    TEXT311 : BOOL ;	//TEXT N.311
    TEXT312 : BOOL ;	//TEXT N.312
    TEXT329 : BOOL ;	//TEXT N.329
    TEXT330 : BOOL ;	//TEXT N.330
    TEXT331 : BOOL ;	//TEXT N.331
    TEXT332 : BOOL ;	//TEXT N.332
    TEXT333 : BOOL ;	//TEXT N.333
    TEXT334 : BOOL ;	//TEXT N.334
    TEXT335 : BOOL ;	//TEXT N.335
    TEXT336 : BOOL ;	//TEXT N.336
    TEXT321 : BOOL ;	//TEXT N.321
    TEXT322 : BOOL ;	//TEXT N.322
    TEXT323 : BOOL ;	//TEXT N.323
    TEXT324 : BOOL ;	//TEXT N.324
    TEXT325 : BOOL ;	//TEXT N.325
    TEXT326 : BOOL ;	//TEXT N.326
    TEXT327 : BOOL ;	//TEXT N.327
    TEXT328 : BOOL ;	//TEXT N.328
    TEXT345 : BOOL ;	//TEXT N.345
    TEXT346 : BOOL ;	//TEXT N.346
    TEXT347 : BOOL ;	//TEXT N.347
    TEXT348 : BOOL ;	//TEXT N.348
    TEXT349 : BOOL ;	//TEXT N.349
    TEXT350 : BOOL ;	//TEXT N.350
    TEXT351 : BOOL ;	//TEXT N.351
    TEXT352 : BOOL ;	//TEXT N.352
    TEXT337 : BOOL ;	//TEXT N.337
    TEXT338 : BOOL ;	//TEXT N.338
    TEXT339 : BOOL ;	//TEXT N.339
    TEXT340 : BOOL ;	//TEXT N.340
    TEXT341 : BOOL ;	//TEXT N.341
    TEXT342 : BOOL ;	//TEXT N.342
    TEXT343 : BOOL ;	//TEXT N.343
    TEXT344 : BOOL ;	//TEXT N.344
    TEXT361 : BOOL ;	//TEXT N.361
    TEXT362 : BOOL ;	//TEXT N.362
    TEXT363 : BOOL ;	//TEXT N.363
    TEXT364 : BOOL ;	//TEXT N.364
    TEXT365 : BOOL ;	//TEXT N.365
    TEXT366 : BOOL ;	//TEXT N.366
    TEXT367 : BOOL ;	//TEXT N.367
    TEXT368 : BOOL ;	//TEXT N.368
    TEXT353 : BOOL ;	//TEXT N.353
    TEXT354 : BOOL ;	//TEXT N.354
    TEXT355 : BOOL ;	//TEXT N.355
    TEXT356 : BOOL ;	//TEXT N.356
    TEXT357 : BOOL ;	//TEXT N.357
    TEXT358 : BOOL ;	//TEXT N.358
    TEXT359 : BOOL ;	//TEXT N.359
    TEXT360 : BOOL ;	//TEXT N.360
    TEXT377 : BOOL ;	//TEXT N.377
    TEXT378 : BOOL ;	//TEXT N.378
    TEXT379 : BOOL ;	//TEXT N.379
    TEXT380 : BOOL ;	//TEXT N.380
    TEXT381 : BOOL ;	//TEXT N.381
    TEXT382 : BOOL ;	//TEXT N.382
    TEXT383 : BOOL ;	//TEXT N.383
    TEXT384 : BOOL ;	//TEXT N.384
    TEXT369 : BOOL ;	//TEXT N.369
    TEXT370 : BOOL ;	//TEXT N.370
    TEXT371 : BOOL ;	//TEXT N.371
    TEXT372 : BOOL ;	//TEXT N.372
    TEXT373 : BOOL ;	//TEXT N.373
    TEXT374 : BOOL ;	//TEXT N.374
    TEXT375 : BOOL ;	//TEXT N.375
    TEXT376 : BOOL ;	//TEXT N.376
    TEXT393 : BOOL ;	//TEXT N.393
    TEXT394 : BOOL ;	//TEXT N.394
    TEXT395 : BOOL ;	//TEXT N.395
    TEXT396 : BOOL ;	//TEXT N.396
    TEXT397 : BOOL ;	//TEXT N.397
    TEXT398 : BOOL ;	//TEXT N.398
    TEXT399 : BOOL ;	//TEXT N.399
    TEXT400 : BOOL ;	//TEXT N.400
    TEXT385 : BOOL ;	//TEXT N.385
    TEXT386 : BOOL ;	//TEXT N.386
    TEXT387 : BOOL ;	//TEXT N.387
    TEXT388 : BOOL ;	//TEXT N.388
    TEXT389 : BOOL ;	//TEXT N.389
    TEXT390 : BOOL ;	//TEXT N.390
    TEXT391 : BOOL ;	//TEXT N.391
    TEXT392 : BOOL ;	//TEXT N.392
    TEXT409 : BOOL ;	//TEXT N.409
    TEXT410 : BOOL ;	//TEXT N.410
    TEXT411 : BOOL ;	//TEXT N.411
    TEXT412 : BOOL ;	//TEXT N.412
    TEXT413 : BOOL ;	//TEXT N.413
    TEXT414 : BOOL ;	//TEXT N.414
    TEXT415 : BOOL ;	//TEXT N.415
    TEXT416 : BOOL ;	//TEXT N.416
    TEXT401 : BOOL ;	//TEXT N.401
    TEXT402 : BOOL ;	//TEXT N.402
    TEXT403 : BOOL ;	//TEXT N.403
    TEXT404 : BOOL ;	//TEXT N.404
    TEXT405 : BOOL ;	//TEXT N.405
    TEXT406 : BOOL ;	//TEXT N.406
    TEXT407 : BOOL ;	//TEXT N.407
    TEXT408 : BOOL ;	//TEXT N.408
    TEXT425 : BOOL ;	//TEXT N.425
    TEXT426 : BOOL ;	//TEXT N.426
    TEXT427 : BOOL ;	//TEXT N.427
    TEXT428 : BOOL ;	//TEXT N.428
    TEXT429 : BOOL ;	//TEXT N.429
    TEXT430 : BOOL ;	//TEXT N.430
    TEXT431 : BOOL ;	//TEXT N.431
    TEXT432 : BOOL ;	//TEXT N.432
    TEXT417 : BOOL ;	//TEXT N.417
    TEXT418 : BOOL ;	//TEXT N.418
    TEXT419 : BOOL ;	//TEXT N.419
    TEXT420 : BOOL ;	//TEXT N.420
    TEXT421 : BOOL ;	//TEXT N.421
    TEXT422 : BOOL ;	//TEXT N.422
    TEXT423 : BOOL ;	//TEXT N.423
    TEXT424 : BOOL ;	//TEXT N.424
    TEXT441 : BOOL ;	//TEXT N.441
    TEXT442 : BOOL ;	//TEXT N.442
    TEXT443 : BOOL ;	//TEXT N.443
    TEXT444 : BOOL ;	//TEXT N.444
    TEXT445 : BOOL ;	//TEXT N.445
    TEXT446 : BOOL ;	//TEXT N.446
    TEXT447 : BOOL ;	//TEXT N.447
    TEXT448 : BOOL ;	//TEXT N.448
    TEXT433 : BOOL ;	//TEXT N.433
    TEXT434 : BOOL ;	//TEXT N.434
    TEXT435 : BOOL ;	//TEXT N.435
    TEXT436 : BOOL ;	//TEXT N.436
    TEXT437 : BOOL ;	//TEXT N.437
    TEXT438 : BOOL ;	//TEXT N.438
    TEXT439 : BOOL ;	//TEXT N.439
    TEXT440 : BOOL ;	//TEXT N.440
    TEXT457 : BOOL ;	//TEXT N.457
    TEXT458 : BOOL ;	//TEXT N.458
    TEXT459 : BOOL ;	//TEXT N.459
    TEXT460 : BOOL ;	//TEXT N.460
    TEXT461 : BOOL ;	//TEXT N.461
    TEXT462 : BOOL ;	//TEXT N.462
    TEXT463 : BOOL ;	//TEXT N.463
    TEXT464 : BOOL ;	//TEXT N.464
    TEXT449 : BOOL ;	//TEXT N.449
    TEXT450 : BOOL ;	//TEXT N.450
    TEXT451 : BOOL ;	//TEXT N.451
    TEXT452 : BOOL ;	//TEXT N.452
    TEXT453 : BOOL ;	//TEXT N.453
    TEXT454 : BOOL ;	//TEXT N.454
    TEXT455 : BOOL ;	//TEXT N.455
    TEXT456 : BOOL ;	//TEXT N.456
    TEXT473 : BOOL ;	//TEXT N.473
    TEXT474 : BOOL ;	//TEXT N.474
    TEXT475 : BOOL ;	//TEXT N.475
    TEXT476 : BOOL ;	//TEXT N.476
    TEXT477 : BOOL ;	//TEXT N.477
    TEXT478 : BOOL ;	//TEXT N.478
    TEXT479 : BOOL ;	//TEXT N.479
    TEXT480 : BOOL ;	//TEXT N.480
    TEXT465 : BOOL ;	//TEXT N.465
    TEXT466 : BOOL ;	//TEXT N.466
    TEXT467 : BOOL ;	//TEXT N.467
    TEXT468 : BOOL ;	//TEXT N.468
    TEXT469 : BOOL ;	//TEXT N.469
    TEXT470 : BOOL ;	//TEXT N.470
    TEXT471 : BOOL ;	//TEXT N.471
    TEXT472 : BOOL ;	//TEXT N.472
    TEXT489 : BOOL ;	//TEXT N.489
    TEXT490 : BOOL ;	//TEXT N.490
    TEXT491 : BOOL ;	//TEXT N.491
    TEXT492 : BOOL ;	//TEXT N.492
    TEXT493 : BOOL ;	//TEXT N.493
    TEXT494 : BOOL ;	//TEXT N.494
    TEXT495 : BOOL ;	//TEXT N.495
    TEXT496 : BOOL ;	//TEXT N.496
    TEXT481 : BOOL ;	//TEXT N.481
    TEXT482 : BOOL ;	//TEXT N.482
    TEXT483 : BOOL ;	//TEXT N.483
    TEXT484 : BOOL ;	//TEXT N.484
    TEXT485 : BOOL ;	//TEXT N.485
    TEXT486 : BOOL ;	//TEXT N.486
    TEXT487 : BOOL ;	//TEXT N.487
    TEXT488 : BOOL ;	//TEXT N.488
    TEXT505 : BOOL ;	//TEXT N.505
    TEXT506 : BOOL ;	//TEXT N.506
    TEXT507 : BOOL ;	//TEXT N.507
    TEXT508 : BOOL ;	//TEXT N.508
    TEXT509 : BOOL ;	//TEXT N.509
    TEXT510 : BOOL ;	//TEXT N.510
    TEXT511 : BOOL ;	//TEXT N.511
    TEXT512 : BOOL ;	//TEXT N.512
    TEXT497 : BOOL ;	//TEXT N.497
    TEXT498 : BOOL ;	//TEXT N.498
    TEXT499 : BOOL ;	//TEXT N.499
    TEXT500 : BOOL ;	//TEXT N.500
    TEXT501 : BOOL ;	//TEXT N.501
    TEXT502 : BOOL ;	//TEXT N.502
    TEXT503 : BOOL ;	//TEXT N.503
    TEXT504 : BOOL ;	//TEXT N.504
    TEXT521 : BOOL ;	//TEXT N.521
    TEXT522 : BOOL ;	//TEXT N.522
    TEXT523 : BOOL ;	//TEXT N.523
    TEXT524 : BOOL ;	//TEXT N.524
    TEXT525 : BOOL ;	//TEXT N.525
    TEXT526 : BOOL ;	//TEXT N.526
    TEXT527 : BOOL ;	//TEXT N.527
    TEXT528 : BOOL ;	//TEXT N.528
    TEXT513 : BOOL ;	//TEXT N.513
    TEXT514 : BOOL ;	//TEXT N.514
    TEXT515 : BOOL ;	//TEXT N.515
    TEXT516 : BOOL ;	//TEXT N.516
    TEXT517 : BOOL ;	//TEXT N.517
    TEXT518 : BOOL ;	//TEXT N.518
    TEXT519 : BOOL ;	//TEXT N.519
    TEXT520 : BOOL ;	//TEXT N.520
    TEXT537 : BOOL ;	//TEXT N.537
    TEXT538 : BOOL ;	//TEXT N.538
    TEXT539 : BOOL ;	//TEXT N.539
    TEXT540 : BOOL ;	//TEXT N.540
    TEXT541 : BOOL ;	//TEXT N.541
    TEXT542 : BOOL ;	//TEXT N.542
    TEXT543 : BOOL ;	//TEXT N.543
    TEXT544 : BOOL ;	//TEXT N.544
    TEXT529 : BOOL ;	//TEXT N.529
    TEXT530 : BOOL ;	//TEXT N.530
    TEXT531 : BOOL ;	//TEXT N.531
    TEXT532 : BOOL ;	//TEXT N.532
    TEXT533 : BOOL ;	//TEXT N.533
    TEXT534 : BOOL ;	//TEXT N.534
    TEXT535 : BOOL ;	//TEXT N.535
    TEXT536 : BOOL ;	//TEXT N.536
    TEXT553 : BOOL ;	//TEXT N.553
    TEXT554 : BOOL ;	//TEXT N.554
    TEXT555 : BOOL ;	//TEXT N.555
    TEXT556 : BOOL ;	//TEXT N.556
    TEXT557 : BOOL ;	//TEXT N.557
    TEXT558 : BOOL ;	//TEXT N.558
    TEXT559 : BOOL ;	//TEXT N.559
    TEXT560 : BOOL ;	//TEXT N.560
    TEXT545 : BOOL ;	//TEXT N.545
    TEXT546 : BOOL ;	//TEXT N.546
    TEXT547 : BOOL ;	//TEXT N.547
    TEXT548 : BOOL ;	//TEXT N.548
    TEXT549 : BOOL ;	//TEXT N.549
    TEXT550 : BOOL ;	//TEXT N.550
    TEXT551 : BOOL ;	//TEXT N.551
    TEXT552 : BOOL ;	//TEXT N.552
    TEXT569 : BOOL ;	//TEXT N.569
    TEXT570 : BOOL ;	//TEXT N.570
    TEXT571 : BOOL ;	//TEXT N.571
    TEXT572 : BOOL ;	//TEXT N.572
    TEXT573 : BOOL ;	//TEXT N.573
    TEXT574 : BOOL ;	//TEXT N.574
    TEXT575 : BOOL ;	//TEXT N.575
    TEXT576 : BOOL ;	//TEXT N.576
    TEXT561 : BOOL ;	//TEXT N.561
    TEXT562 : BOOL ;	//TEXT N.562
    TEXT563 : BOOL ;	//TEXT N.563
    TEXT564 : BOOL ;	//TEXT N.564
    TEXT565 : BOOL ;	//TEXT N.565
    TEXT566 : BOOL ;	//TEXT N.566
    TEXT567 : BOOL ;	//TEXT N.567
    TEXT568 : BOOL ;	//TEXT N.568
    TEXT585 : BOOL ;	//TEXT N.585
    TEXT586 : BOOL ;	//TEXT N.586
    TEXT587 : BOOL ;	//TEXT N.587
    TEXT588 : BOOL ;	//TEXT N.588
    TEXT589 : BOOL ;	//TEXT N.589
    TEXT590 : BOOL ;	//TEXT N.590
    TEXT591 : BOOL ;	//TEXT N.591
    TEXT592 : BOOL ;	//TEXT N.592
    TEXT577 : BOOL ;	//TEXT N.577
    TEXT578 : BOOL ;	//TEXT N.578
    TEXT579 : BOOL ;	//TEXT N.579
    TEXT580 : BOOL ;	//TEXT N.580
    TEXT581 : BOOL ;	//TEXT N.581
    TEXT582 : BOOL ;	//TEXT N.582
    TEXT583 : BOOL ;	//TEXT N.583
    TEXT584 : BOOL ;	//TEXT N.584
    TEXT601 : BOOL ;	//TEXT N.601
    TEXT602 : BOOL ;	//TEXT N.602
    TEXT603 : BOOL ;	//TEXT N.603
    TEXT604 : BOOL ;	//TEXT N.604
    TEXT605 : BOOL ;	//TEXT N.605
    TEXT606 : BOOL ;	//TEXT N.606
    TEXT607 : BOOL ;	//TEXT N.607
    TEXT608 : BOOL ;	//TEXT N.608
    TEXT593 : BOOL ;	//TEXT N.593
    TEXT594 : BOOL ;	//TEXT N.594
    TEXT595 : BOOL ;	//TEXT N.595
    TEXT596 : BOOL ;	//TEXT N.596
    TEXT597 : BOOL ;	//TEXT N.597
    TEXT598 : BOOL ;	//TEXT N.598
    TEXT599 : BOOL ;	//TEXT N.599
    TEXT600 : BOOL ;	//TEXT N.600
    TEXT617 : BOOL ;	//TEXT N.617
    TEXT618 : BOOL ;	//TEXT N.618
    TEXT619 : BOOL ;	//TEXT N.619
    TEXT620 : BOOL ;	//TEXT N.620
    TEXT621 : BOOL ;	//TEXT N.621
    TEXT622 : BOOL ;	//TEXT N.622
    TEXT623 : BOOL ;	//TEXT N.623
    TEXT624 : BOOL ;	//TEXT N.624
    TEXT609 : BOOL ;	//TEXT N.609
    TEXT610 : BOOL ;	//TEXT N.610
    TEXT611 : BOOL ;	//TEXT N.611
    TEXT612 : BOOL ;	//TEXT N.612
    TEXT613 : BOOL ;	//TEXT N.613
    TEXT614 : BOOL ;	//TEXT N.614
    TEXT615 : BOOL ;	//TEXT N.615
    TEXT616 : BOOL ;	//TEXT N.616
    TEXT633 : BOOL ;	//TEXT N.633
    TEXT634 : BOOL ;	//TEXT N.634
    TEXT635 : BOOL ;	//TEXT N.635
    TEXT636 : BOOL ;	//TEXT N.636
    TEXT637 : BOOL ;	//TEXT N.637
    TEXT638 : BOOL ;	//TEXT N.638
    TEXT639 : BOOL ;	//TEXT N.639
    TEXT640 : BOOL ;	//TEXT N.640
    TEXT625 : BOOL ;	//TEXT N.625
    TEXT626 : BOOL ;	//TEXT N.626
    TEXT627 : BOOL ;	//TEXT N.627
    TEXT628 : BOOL ;	//TEXT N.628
    TEXT629 : BOOL ;	//TEXT N.629
    TEXT630 : BOOL ;	//TEXT N.630
    TEXT631 : BOOL ;	//TEXT N.631
    TEXT632 : BOOL ;	//TEXT N.632
   END_STRUCT ;
   PaginaDaVisualizzare : INT ;	//Number of page to display
   PaginaPrecedenteSetup : INT ;	//Number of page displayed before "Setup" page
   NumeroComandoManuale : INT ;	//Number of manual command
   BoschProgramManuale : BYTE ;	//Number of program of screwdriver in manual mode
   ServiceAsseSelezionato : BYTE ;	//Axis selected for movement in service mode (0=X; 1=Y; 2=Z; 3=C; 4=P)
   ServiceTipoJog : BYTE ;	//Kind of jog movement in service mode (0=continue; 1=incremental)
   ServiceFieldsDisplayed : BYTE ;	//Identify the fields to be displayed in service page
   TypePointTeachIn : BYTE ;	//Kind of screw in teach-in mode
   PointWeldingTeachIn : BYTE ;	//Identification of the screw in tech-in mode
   TeachInFieldsDisplayed : STRUCT 	//Identify the fields to be displayed in teach-in page
    Punto1Saldatura : BOOL ;
    Punto2Saldatura : BOOL ;
    Punto3Saldatura : BOOL ;
    Punto4Saldatura : BOOL ;
    Punto5Saldatura : BOOL ;
    Punto6Saldatura : BOOL ;
    Punto7Saldatura : BOOL ;
    Punto8Saldatura : BOOL ;
    Punto9Saldatura : BOOL ;
    Punto10Saldatura : BOOL ;
    Punto11Saldatura : BOOL ;
    Punto12Saldatura : BOOL ;
    Punto13Saldatura : BOOL ;
    PuntoVisione : BOOL ;
    Riserva1 : BOOL ;
    Riserva2 : BOOL ;
   END_STRUCT ;
   Target_Inc : DINT ;	//Target for the incremental movement
  END_STRUCT ;	
BEGIN
END_DATA_BLOCK

DATA_BLOCK "Timer"	// DB 20
VERSION : 0.1
  STRUCT
   TmrOutGas : S5TIME  := S5T#1M;
   TmrIgnition : S5TIME  := S5T#20S;
   TmrDelayWelding : S5TIME  := S5T#300MS;
   time1 : S5TIME ;
   time11 : S5TIME ;
   time12 : S5TIME ;
   time13 : S5TIME ;
   time14 : S5TIME ;
   time15 : S5TIME ;
   time16 : S5TIME ;
   time17 : S5TIME ;
   time18 : S5TIME ;
   time19 : S5TIME ;
   time110 : S5TIME ;
   time111 : S5TIME ;
   time112 : S5TIME ;
   time113 : S5TIME ;
   time114 : S5TIME ;
   time115 : S5TIME ;
   time116 : S5TIME ;
   Override : INT  := 20;
   riserva : INT ;
   riserva2 : INT ;
   Comp01_OK : BOOL ;
   Comp02_OK : BOOL ;
   Comp03_OK : BOOL ;
   Comp04_OK : BOOL ;
   Comp05_OK : BOOL ;
   Comp06_OK : BOOL ;
   Comp07_OK : BOOL ;
   Comp08_OK : BOOL ;
   Comp09_OK : BOOL ;
   Comp10_OK : BOOL ;
   Comp11_OK : BOOL ;
   Comp12_OK : BOOL ;
   Comp13_OK : BOOL ;
   Comp14_OK : BOOL ;
   Comp15_OK : BOOL ;
   Comp16_OK : BOOL ;
   OffsetX : DINT ;
   OffsetY : DINT ;
   okAletta1 : BOOL ;
   okAletta2 : BOOL ;
   okAletta3 : BOOL ;
   okAletta4 : BOOL ;
   okAletta5 : BOOL ;
   okAletta6 : BOOL ;
   okAletta7 : BOOL ;
   okAletta8 : BOOL ;
   okAletta9 : BOOL ;
   okAletta10 : BOOL ;
   okAletta11 : BOOL ;
   okAletta12 : BOOL ;
   okAletta13 : BOOL ;
   okAletta14 : BOOL ;
   okAletta15 : BOOL ;
   okAletta16 : BOOL ;
   okAletta17 : BOOL ;
   okAletta18 : BOOL ;
   okAletta19 : BOOL ;
   okAletta20 : BOOL ;
   CheckComponent : BOOL  := TRUE;	//Check component with tool 1 --> Disable ; 0 --> Enable
   CheckTelec : BOOL ;	//Check Component with Omron 1 --> Disable ; 0 --> Enable
   Check1 : BOOL ;
   Check2 : BOOL ;
   okAletta1_PP : BOOL ;
   okAletta2_PP : BOOL ;
   okAletta3_PP : BOOL ;
   okAletta4_PP : BOOL ;
   okAletta5_PP : BOOL ;
   okAletta6_PP : BOOL ;
   okAletta7_PP : BOOL ;
   okAletta8_PP : BOOL ;
   okAletta9_PP : BOOL ;
   okAletta10_PP : BOOL ;
   okAletta11_PP : BOOL ;
   okAletta12_PP : BOOL ;
   okAletta13_PP : BOOL ;
   okAletta14_PP : BOOL ;
   okAletta15_PP : BOOL ;
   okAletta16_PP : BOOL ;
   okAletta17_PP : BOOL ;
   okAletta18_PP : BOOL ;
   okAletta19_PP : BOOL ;
   okAletta20_PP : BOOL ;
   NumberVane : INT ;
  END_STRUCT ;	
BEGIN
   TmrOutGas := S5T#1M;
   TmrIgnition := S5T#20S;
   TmrDelayWelding := S5T#300MS;
   Override := 100;
   OffsetX := L#350;
   OffsetY := L#400;
END_DATA_BLOCK

DATA_BLOCK "DBWork"	// DB 21
TITLE = Recipe of part in production
AUTHOR : Coletti
VERSION : 0.1
  STRUCT
   Famiglia : BYTE  := B#16#2;	//Type of family of product(2=Step2; 3=Step3)
   Turbo : BYTE  := B#16#1;	//Type of product
   Portapezzo1 : INT  := 1;	//Code of work rest 1
   Portapezzo2 : INT  := 1;	//Code of work rest 2
   TempoSaldatura : ARRAY  [1 .. 20 ] OF STRUCT
    Tempo : S5TIME  := S5T#1S;
   END_STRUCT ;
   CoordSaldatura : ARRAY  [1 .. 20 ] OF //Coordinates of points
   STRUCT
    X1 : DINT ;	//X coordinate of point
    Y1 : DINT ;	//Y coordinate of point
    X2 : DINT ;
    Y2 : DINT ;
   END_STRUCT ;
   EnableTelecamera : BOOL  := TRUE;
   PP : ARRAY  [1 .. 2 ] OF STRUCT
    Vuoto : BOOL ;
    Caricato : BOOL ;
    Bloccato : BOOL ;
    Fuori : BOOL ;
    Dentro : BOOL ;
    InLavorazione : BOOL ;
    Lavorato : BOOL ;
    Buono : BOOL ;
    Scarto : BOOL ;
    NumSaldaturaAtt : INT ;
   END_STRUCT ;
   NumeroAnomalie : DINT ;
   NumeroPezziProd : DINT ;
   NumeroSaldature : INT ;
   Riserva : DINT ;	//position X for camera check
   Riserva1 : DINT ;	//position Y for camera check
   RotationTable : BOOL ;	//angle rotation 1-->PP1 on welding; 0-->PP2 on Welding
   PointCamCheck : ARRAY  [1 .. 10 ] OF STRUCT
    x : DINT ;
    y : DINT ;
   END_STRUCT ;
  END_STRUCT ;	
BEGIN
   Famiglia := B#16#2;
   Turbo := B#16#1;
   Portapezzo1 := 1;
   Portapezzo2 := 1;
   TempoSaldatura[1].Tempo := S5T#1S;
   TempoSaldatura[2].Tempo := S5T#2S;
   TempoSaldatura[3].Tempo := S5T#1S;
   TempoSaldatura[4].Tempo := S5T#1S;
   TempoSaldatura[5].Tempo := S5T#1S;
   TempoSaldatura[6].Tempo := S5T#1S;
   TempoSaldatura[7].Tempo := S5T#1S;
   TempoSaldatura[8].Tempo := S5T#1S;
   TempoSaldatura[9].Tempo := S5T#1S;
   TempoSaldatura[10].Tempo := S5T#1S;
   TempoSaldatura[11].Tempo := S5T#1S;
   TempoSaldatura[12].Tempo := S5T#1S;
   TempoSaldatura[13].Tempo := S5T#1S;
   TempoSaldatura[14].Tempo := S5T#1S;
   TempoSaldatura[15].Tempo := S5T#1S;
   TempoSaldatura[16].Tempo := S5T#1S;
   TempoSaldatura[17].Tempo := S5T#1S;
   TempoSaldatura[18].Tempo := S5T#1S;
   TempoSaldatura[19].Tempo := S5T#1S;
   TempoSaldatura[20].Tempo := S5T#1S;
   CoordSaldatura[1].X1 := L#-60766;
   CoordSaldatura[1].Y1 := L#-86096;
   CoordSaldatura[1].X2 := L#-60406;
   CoordSaldatura[1].Y2 := L#-86246;
   CoordSaldatura[2].X1 := L#-46600;
   CoordSaldatura[2].Y1 := L#-81431;
   CoordSaldatura[2].X2 := L#-46422;
   CoordSaldatura[2].Y2 := L#-81523;
   CoordSaldatura[3].X1 := L#-29709;
   CoordSaldatura[3].Y1 := L#-81739;
   CoordSaldatura[3].X2 := L#-29405;
   CoordSaldatura[3].Y2 := L#-81809;
   CoordSaldatura[4].X1 := L#-16402;
   CoordSaldatura[4].Y1 := L#-86931;
   CoordSaldatura[4].X2 := L#-116220;
   CoordSaldatura[4].Y2 := L#-86961;
   CoordSaldatura[5].X1 := L#-11762;
   CoordSaldatura[5].Y1 := L#-95066;
   CoordSaldatura[5].X2 := L#-11500;
   CoordSaldatura[5].Y2 := L#-95199;
   CoordSaldatura[6].X1 := L#-17500;
   CoordSaldatura[6].Y1 := L#-102971;
   CoordSaldatura[6].X2 := L#-17415;
   CoordSaldatura[6].Y2 := L#-103088;
   CoordSaldatura[7].X1 := L#-31505;
   CoordSaldatura[7].Y1 := L#-107714;
   CoordSaldatura[7].X2 := L#-31400;
   CoordSaldatura[7].Y2 := L#-108200;
   CoordSaldatura[8].X1 := L#-48449;
   CoordSaldatura[8].Y1 := L#-107375;
   CoordSaldatura[8].X2 := L#-48367;
   CoordSaldatura[8].Y2 := L#-107501;
   CoordSaldatura[9].X1 := L#-61760;
   CoordSaldatura[9].Y1 := L#-102188;
   CoordSaldatura[9].X2 := L#-61561;
   CoordSaldatura[9].Y2 := L#-102300;
   CoordSaldatura[10].X1 := L#-66400;
   CoordSaldatura[10].Y1 := L#-94028;
   CoordSaldatura[10].Y2 := L#-94249;
   EnableTelecamera := TRUE;
END_DATA_BLOCK

DATA_BLOCK "coordinate"	// DB 22
VERSION : 0.1
  STRUCT
   CoordSaldaturaPP1 : ARRAY  [1 .. 20 ] OF //Coordinates of points
   STRUCT
    X1 : DINT ;	//X coordinate of point PP1
    Y1 : DINT ;	//Y coordinate of point PP1
    X2 : DINT ;
    Y2 : DINT ;
   END_STRUCT ;
   CoordSaldaturaPP2 : ARRAY  [1 .. 20 ] OF //Coordinates of points
   STRUCT
    X1 : DINT ;	//X coordinate of point PP2
    Y1 : DINT ;	//Y coordinate of point PP2
    X2 : DINT ;
    Y2 : DINT ;
   END_STRUCT ;
   CoordSaldaturaPP3 : ARRAY  [1 .. 20 ] OF //Coordinates of points
   STRUCT
    X1 : DINT ;	//X coordinate of point PP3
    Y1 : DINT ;	//Y coordinate of point PP3
    X2 : DINT ;
    Y2 : DINT ;
   END_STRUCT ;
   CoordSaldaturaPP4 : ARRAY  [1 .. 20 ] OF //Coordinates of points
   STRUCT
    X1 : DINT ;	//X coordinate of point PP4
    Y1 : DINT ;	//Y coordinate of point PP4
    X2 : DINT ;
    Y2 : DINT ;
   END_STRUCT ;
   CoordSaldaturaPP5 : ARRAY  [1 .. 20 ] OF //Coordinates of points
   STRUCT
    X1 : DINT ;	//X coordinate of point PP5
    Y1 : DINT ;	//Y coordinate of point PP5
    X2 : DINT ;
    Y2 : DINT ;
   END_STRUCT ;
   CoordSaldaturaPP6 : ARRAY  [1 .. 20 ] OF STRUCT
    X1 : DINT ;
    Y1 : DINT ;
    X2 : DINT ;
    Y2 : DINT ;
   END_STRUCT ;
   CoordSaldaturaPP7 : ARRAY  [1 .. 20 ] OF STRUCT
    X1 : DINT ;
    Y1 : DINT ;
    X2 : DINT ;
    Y2 : DINT ;
   END_STRUCT ;
   CoordSaldaturaPP8 : ARRAY  [1 .. 20 ] OF STRUCT
    X1 : DINT ;
    Y1 : DINT ;
    X2 : DINT ;
    Y2 : DINT ;
   END_STRUCT ;
   CoordSaldaturaPP9 : ARRAY  [1 .. 20 ] OF STRUCT
    X1 : DINT ;
    Y1 : DINT ;
    X2 : DINT ;
    Y2 : DINT ;
   END_STRUCT ;
   CoordSaldaturaPP10 : ARRAY  [1 .. 20 ] OF STRUCT
    X1 : DINT ;
    Y1 : DINT ;
    X2 : DINT ;
    Y2 : DINT ;
   END_STRUCT ;
   CoordSaldaturaPP11 : ARRAY  [1 .. 20 ] OF STRUCT
    X1 : DINT ;
    Y1 : DINT ;
    X2 : DINT ;
    Y2 : DINT ;
   END_STRUCT ;
   CoordSaldaturaPP12 : ARRAY  [1 .. 20 ] OF STRUCT
    X1 : DINT ;
    Y1 : DINT ;
    X2 : DINT ;
    Y2 : DINT ;
   END_STRUCT ;
   CoordSaldaturaPP13 : ARRAY  [1 .. 20 ] OF STRUCT
    X1 : DINT ;
    Y1 : DINT ;
    X2 : DINT ;
    Y2 : DINT ;
   END_STRUCT ;
   CoordSaldaturaPP14 : ARRAY  [1 .. 20 ] OF STRUCT
    X1 : DINT ;
    Y1 : DINT ;
    X2 : DINT ;
    Y2 : DINT ;
   END_STRUCT ;
   CoordSaldaturaPP15 : ARRAY  [1 .. 20 ] OF STRUCT
    X1 : DINT ;
    Y1 : DINT ;
    X2 : DINT ;
    Y2 : DINT ;
   END_STRUCT ;
   CoordSaldaturaPP16 : ARRAY  [1 .. 20 ] OF STRUCT
    X1 : DINT ;
    Y1 : DINT ;
    X2 : DINT ;
    Y2 : DINT ;
   END_STRUCT ;
   CoordSaldaturaPP17 : ARRAY  [1 .. 20 ] OF STRUCT
    X1 : DINT ;
    Y1 : DINT ;
    X2 : DINT ;
    Y2 : DINT ;
   END_STRUCT ;
   CoordSaldaturaPP18 : ARRAY  [1 .. 20 ] OF STRUCT
    X1 : DINT ;
    Y1 : DINT ;
    X2 : DINT ;
    Y2 : DINT ;
   END_STRUCT ;
   CoordSaldaturaPP19 : ARRAY  [1 .. 20 ] OF STRUCT
    X1 : DINT ;
    Y1 : DINT ;
    X2 : DINT ;
    Y2 : DINT ;
   END_STRUCT ;
   CoordSaldaturaPP20 : ARRAY  [1 .. 20 ] OF STRUCT
    X1 : DINT ;
    Y1 : DINT ;
    X2 : DINT ;
    Y2 : DINT ;
   END_STRUCT ;
   CoordinateCam_PP1 : ARRAY  [1 .. 10 ] OF STRUCT
    X : DINT ;	//X coordinate of point cam PP1
    Y : DINT ;	//X coordinate of point cam PP1
   END_STRUCT ;
   CoordinateCam_PP2 : ARRAY  [1 .. 10 ] OF STRUCT
    X : DINT ;	//X coordinate of point cam PP1
    Y : DINT ;	//X coordinate of point cam PP1
   END_STRUCT ;
   CoordinateCam_PP3 : ARRAY  [1 .. 10 ] OF STRUCT
    X : DINT ;	//X coordinate of point cam PP1
    Y : DINT ;	//X coordinate of point cam PP1
   END_STRUCT ;
   CoordinateCam_PP4 : ARRAY  [1 .. 10 ] OF STRUCT
    X : DINT ;	//X coordinate of point cam PP1
    Y : DINT ;	//X coordinate of point cam PP1
   END_STRUCT ;
   CoordinateCam_PP5 : ARRAY  [1 .. 10 ] OF STRUCT
    X : DINT ;	//X coordinate of point cam PP1
    Y : DINT ;	//X coordinate of point cam PP1
   END_STRUCT ;
   CoordinateCam_PP6 : ARRAY  [1 .. 10 ] OF STRUCT
    X : DINT ;	//X coordinate of point cam PP1
    Y : DINT ;	//X coordinate of point cam PP1
   END_STRUCT ;
   CoordinateCam_PP7 : ARRAY  [1 .. 10 ] OF STRUCT
    X : DINT ;	//X coordinate of point cam PP1
    Y : DINT ;	//X coordinate of point cam PP1
   END_STRUCT ;
   CoordinateCam_PP8 : ARRAY  [1 .. 10 ] OF STRUCT
    X : DINT ;	//X coordinate of point cam PP1
    Y : DINT ;	//X coordinate of point cam PP1
   END_STRUCT ;
   CoordinateCam_PP9 : ARRAY  [1 .. 10 ] OF STRUCT
    X : DINT ;	//X coordinate of point cam PP1
    Y : DINT ;	//X coordinate of point cam PP1
   END_STRUCT ;
   CoordinateCam_PP10 : ARRAY  [1 .. 10 ] OF STRUCT
    X : DINT ;	//X coordinate of point cam PP1
    Y : DINT ;	//X coordinate of point cam PP1
   END_STRUCT ;
   CoordinateCam_PP11 : ARRAY  [1 .. 10 ] OF STRUCT
    X : DINT ;	//X coordinate of point cam PP1
    Y : DINT ;	//X coordinate of point cam PP1
   END_STRUCT ;
   CoordinateCam_PP12 : ARRAY  [1 .. 10 ] OF STRUCT
    X : DINT ;	//X coordinate of point cam PP1
    Y : DINT ;	//X coordinate of point cam PP1
   END_STRUCT ;
   CoordinateCam_PP13 : ARRAY  [1 .. 10 ] OF STRUCT
    X : DINT ;	//X coordinate of point cam PP1
    Y : DINT ;	//X coordinate of point cam PP1
   END_STRUCT ;
   CoordinateCam_PP14 : ARRAY  [1 .. 10 ] OF STRUCT
    X : DINT ;	//X coordinate of point cam PP1
    Y : DINT ;	//X coordinate of point cam PP1
   END_STRUCT ;
   CoordinateCam_PP15 : ARRAY  [1 .. 10 ] OF STRUCT
    X : DINT ;	//X coordinate of point cam PP1
    Y : DINT ;	//X coordinate of point cam PP1
   END_STRUCT ;
   CoordinateCam_PP16 : ARRAY  [1 .. 10 ] OF STRUCT
    X : DINT ;	//X coordinate of point cam PP1
    Y : DINT ;	//X coordinate of point cam PP1
   END_STRUCT ;
   CoordinateCam_PP17 : ARRAY  [1 .. 10 ] OF STRUCT
    X : DINT ;	//X coordinate of point cam PP1
    Y : DINT ;	//X coordinate of point cam PP1
   END_STRUCT ;
   CoordinateCam_PP18 : ARRAY  [1 .. 10 ] OF STRUCT
    X : DINT ;	//X coordinate of point cam PP1
    Y : DINT ;	//X coordinate of point cam PP1
   END_STRUCT ;
   CoordinateCam_PP19 : ARRAY  [1 .. 10 ] OF STRUCT
    X : DINT ;	//X coordinate of point cam PP1
    Y : DINT ;	//X coordinate of point cam PP1
   END_STRUCT ;
   CoordinateCam_PP20 : ARRAY  [1 .. 10 ] OF STRUCT
    X : DINT ;	//X coordinate of point cam PP1
    Y : DINT ;	//X coordinate of point cam PP1
   END_STRUCT ;
   NumeroSaldaturePP1 : INT ;
   NumeroSaldaturePP2 : INT ;
   NumeroSaldaturePP3 : INT ;
   NumeroSaldaturePP4 : INT ;
   NumeroSaldaturePP5 : INT ;
   NumeroSaldaturePP6 : INT ;
   NumeroSaldaturePP7 : INT ;
   NumeroSaldaturePP8 : INT ;
   NumeroSaldaturePP9 : INT ;
   NumeroSaldaturePP10 : INT ;
   NumeroSaldaturePP11 : INT ;
   NumeroSaldaturePP12 : INT ;
   NumeroSaldaturePP13 : INT ;
   NumeroSaldaturePP14 : INT ;
   NumeroSaldaturePP15 : INT ;
   NumeroSaldaturePP16 : INT ;
   NumeroSaldaturePP17 : INT ;
   NumeroSaldaturePP18 : INT ;
   NumeroSaldaturePP19 : INT ;
   NumeroSaldaturePP20 : INT ;
   TimeWeldingPP1 : ARRAY  [1 .. 20 ] OF STRUCT
    Tempo : S5TIME  := S5T#1S;
   END_STRUCT ;
   TimeWeldingPP2 : ARRAY  [1 .. 20 ] OF STRUCT
    Tempo : S5TIME  := S5T#1S;
   END_STRUCT ;
   TimeWeldingPP3 : ARRAY  [1 .. 20 ] OF STRUCT
    Tempo : S5TIME  := S5T#1S;
   END_STRUCT ;
   TimeWeldingPP4 : ARRAY  [1 .. 20 ] OF STRUCT
    Tempo : S5TIME  := S5T#1S;
   END_STRUCT ;
   TimeWeldingPP5 : ARRAY  [1 .. 20 ] OF STRUCT
    Tempo : S5TIME  := S5T#1S;
   END_STRUCT ;
   TimeWeldingPP6 : ARRAY  [1 .. 20 ] OF STRUCT
    Tempo : S5TIME  := S5T#1S;
   END_STRUCT ;
   TimeWeldingPP7 : ARRAY  [1 .. 20 ] OF STRUCT
    Tempo : S5TIME  := S5T#1S;
   END_STRUCT ;
   TimeWeldingPP8 : ARRAY  [1 .. 20 ] OF STRUCT
    Tempo : S5TIME  := S5T#1S;
   END_STRUCT ;
   TimeWeldingPP9 : ARRAY  [1 .. 20 ] OF STRUCT
    Tempo : S5TIME  := S5T#1S;
   END_STRUCT ;
   TimeWeldingPP10 : ARRAY  [1 .. 20 ] OF STRUCT
    Tempo : S5TIME  := S5T#1S;
   END_STRUCT ;
   TimeWeldingPP11 : ARRAY  [1 .. 20 ] OF STRUCT
    Tempo : S5TIME  := S5T#1S;
   END_STRUCT ;
   TimeWeldingPP12 : ARRAY  [1 .. 20 ] OF STRUCT
    Tempo : S5TIME  := S5T#1S;
   END_STRUCT ;
   TimeWeldingPP13 : ARRAY  [1 .. 20 ] OF STRUCT
    Tempo : S5TIME  := S5T#1S;
   END_STRUCT ;
   TimeWeldingPP14 : ARRAY  [1 .. 20 ] OF STRUCT
    Tempo : S5TIME  := S5T#1S;
   END_STRUCT ;
   TimeWeldingPP15 : ARRAY  [1 .. 20 ] OF STRUCT
    Tempo : S5TIME  := S5T#1S;
   END_STRUCT ;
   TimeWeldingPP16 : ARRAY  [1 .. 20 ] OF STRUCT
    Tempo : S5TIME  := S5T#1S;
   END_STRUCT ;
   TimeWeldingPP17 : ARRAY  [1 .. 20 ] OF STRUCT
    Tempo : S5TIME  := S5T#1S;
   END_STRUCT ;
   TimeWeldingPP18 : ARRAY  [1 .. 20 ] OF STRUCT
    Tempo : S5TIME  := S5T#1S;
   END_STRUCT ;
   TimeWeldingPP19 : ARRAY  [1 .. 20 ] OF STRUCT
    Tempo : S5TIME  := S5T#1S;
   END_STRUCT ;
   TimeWeldingPP20 : ARRAY  [1 .. 20 ] OF STRUCT
    Tempo : S5TIME  := S5T#1S;
   END_STRUCT ;
  END_STRUCT ;	
BEGIN
   CoordSaldaturaPP1[1].X1 := L#-60530;
   CoordSaldaturaPP1[1].Y1 := L#-172340;
   CoordSaldaturaPP1[1].X2 := L#-60530;
   CoordSaldaturaPP1[1].Y2 := L#-172340;
   CoordSaldaturaPP1[2].X1 := L#-46530;
   CoordSaldaturaPP1[2].Y1 := L#-162870;
   CoordSaldaturaPP1[2].X2 := L#-46530;
   CoordSaldaturaPP1[2].Y2 := L#-162870;
   CoordSaldaturaPP1[3].X1 := L#-29630;
   CoordSaldaturaPP1[3].Y1 := L#-163440;
   CoordSaldaturaPP1[3].X2 := L#-29630;
   CoordSaldaturaPP1[3].Y2 := L#-163440;
   CoordSaldaturaPP1[4].X1 := L#-16300;
   CoordSaldaturaPP1[4].Y1 := L#-173820;
   CoordSaldaturaPP1[4].X2 := L#-16300;
   CoordSaldaturaPP1[4].Y2 := L#-173820;
   CoordSaldaturaPP1[5].X1 := L#-11620;
   CoordSaldaturaPP1[5].Y1 := L#-190070;
   CoordSaldaturaPP1[5].X2 := L#-11620;
   CoordSaldaturaPP1[5].Y2 := L#-190070;
   CoordSaldaturaPP1[6].X1 := L#-17370;
   CoordSaldaturaPP1[6].Y1 := L#-205960;
   CoordSaldaturaPP1[6].X2 := L#-17370;
   CoordSaldaturaPP1[6].Y2 := L#-205960;
   CoordSaldaturaPP1[7].X1 := L#-31370;
   CoordSaldaturaPP1[7].Y1 := L#-215430;
   CoordSaldaturaPP1[7].X2 := L#-31370;
   CoordSaldaturaPP1[7].Y2 := L#-215430;
   CoordSaldaturaPP1[8].X1 := L#-48270;
   CoordSaldaturaPP1[8].Y1 := L#-214860;
   CoordSaldaturaPP1[8].X2 := L#-48270;
   CoordSaldaturaPP1[8].Y2 := L#-214860;
   CoordSaldaturaPP1[9].X1 := L#-61600;
   CoordSaldaturaPP1[9].Y1 := L#-204480;
   CoordSaldaturaPP1[9].X2 := L#-61600;
   CoordSaldaturaPP1[9].Y2 := L#-204480;
   CoordSaldaturaPP1[10].X1 := L#-66280;
   CoordSaldaturaPP1[10].Y1 := L#-188230;
   CoordSaldaturaPP1[10].X2 := L#-66280;
   CoordSaldaturaPP1[10].Y2 := L#-188230;
   CoordSaldaturaPP6[1].X1 := L#-24431;
   CoordSaldaturaPP6[1].Y1 := L#-211667;
   CoordSaldaturaPP6[1].X2 := L#-24468;
   CoordSaldaturaPP6[1].Y2 := L#-211634;
   CoordSaldaturaPP6[2].X1 := L#-13011;
   CoordSaldaturaPP6[2].Y1 := L#-199436;
   CoordSaldaturaPP6[2].X2 := L#-12856;
   CoordSaldaturaPP6[2].Y2 := L#-199488;
   CoordSaldaturaPP6[3].X1 := L#-9745;
   CoordSaldaturaPP6[3].Y1 := L#-183598;
   CoordSaldaturaPP6[3].X2 := L#-9756;
   CoordSaldaturaPP6[3].Y2 := L#-183663;
   CoordSaldaturaPP6[4].X1 := L#-16203;
   CoordSaldaturaPP6[4].Y1 := L#-168150;
   CoordSaldaturaPP6[4].X2 := L#-16141;
   CoordSaldaturaPP6[4].Y2 := L#-168156;
   CoordSaldaturaPP6[5].X1 := L#-29434;
   CoordSaldaturaPP6[5].Y1 := L#-158429;
   CoordSaldaturaPP6[5].X2 := L#-29472;
   CoordSaldaturaPP6[5].Y2 := L#-158489;
   CoordSaldaturaPP6[6].X1 := L#-46262;
   CoordSaldaturaPP6[6].Y1 := L#-157658;
   CoordSaldaturaPP6[6].X2 := L#-46155;
   CoordSaldaturaPP6[6].Y2 := L#-157716;
   CoordSaldaturaPP6[7].X1 := L#-60740;
   CoordSaldaturaPP6[7].Y1 := L#-166127;
   CoordSaldaturaPP6[7].X2 := L#-60564;
   CoordSaldaturaPP6[7].Y2 := L#-166296;
   CoordSaldaturaPP6[8].X1 := L#-68335;
   CoordSaldaturaPP6[8].Y1 := L#-180765;
   CoordSaldaturaPP6[8].X2 := L#-68026;
   CoordSaldaturaPP6[8].Y2 := L#-180787;
   CoordSaldaturaPP6[9].X1 := L#-66468;
   CoordSaldaturaPP6[9].Y1 := L#-197254;
   CoordSaldaturaPP6[9].X2 := L#-66217;
   CoordSaldaturaPP6[9].Y2 := L#-197398;
   CoordSaldaturaPP6[10].X1 := L#-56162;
   CoordSaldaturaPP6[10].Y1 := L#-210332;
   CoordSaldaturaPP6[10].X2 := L#-56200;
   CoordSaldaturaPP6[10].Y2 := L#-210331;
   CoordSaldaturaPP6[11].X1 := L#-40981;
   CoordSaldaturaPP6[11].Y1 := L#-215911;
   CoordSaldaturaPP6[11].X2 := L#-40587;
   CoordSaldaturaPP6[11].Y2 := L#-215681;
   CoordSaldaturaPP11[1].X1 := L#-24431;
   CoordSaldaturaPP11[1].Y1 := L#-211667;
   CoordSaldaturaPP11[1].X2 := L#-24468;
   CoordSaldaturaPP11[1].Y2 := L#-211634;
   CoordSaldaturaPP11[2].X1 := L#-13011;
   CoordSaldaturaPP11[2].Y1 := L#-199436;
   CoordSaldaturaPP11[2].X2 := L#-12856;
   CoordSaldaturaPP11[2].Y2 := L#-199488;
   CoordSaldaturaPP11[3].X1 := L#-9745;
   CoordSaldaturaPP11[3].Y1 := L#-183598;
   CoordSaldaturaPP11[3].X2 := L#-9786;
   CoordSaldaturaPP11[3].Y2 := L#-183663;
   CoordSaldaturaPP11[4].X1 := L#-16203;
   CoordSaldaturaPP11[4].Y1 := L#-168150;
   CoordSaldaturaPP11[4].X2 := L#-16141;
   CoordSaldaturaPP11[4].Y2 := L#-168156;
   CoordSaldaturaPP11[5].X1 := L#-29434;
   CoordSaldaturaPP11[5].Y1 := L#-158429;
   CoordSaldaturaPP11[5].X2 := L#-29472;
   CoordSaldaturaPP11[5].Y2 := L#-158489;
   CoordSaldaturaPP11[6].X1 := L#-46262;
   CoordSaldaturaPP11[6].Y1 := L#-157658;
   CoordSaldaturaPP11[6].X2 := L#-46155;
   CoordSaldaturaPP11[6].Y2 := L#-157716;
   CoordSaldaturaPP11[7].X1 := L#-60740;
   CoordSaldaturaPP11[7].Y1 := L#-166127;
   CoordSaldaturaPP11[7].X2 := L#-60564;
   CoordSaldaturaPP11[7].Y2 := L#-166296;
   CoordSaldaturaPP11[8].X1 := L#-68335;
   CoordSaldaturaPP11[8].Y1 := L#-180765;
   CoordSaldaturaPP11[8].X2 := L#-68026;
   CoordSaldaturaPP11[8].Y2 := L#-180787;
   CoordSaldaturaPP11[9].X1 := L#-66468;
   CoordSaldaturaPP11[9].Y1 := L#-197254;
   CoordSaldaturaPP11[9].X2 := L#-66217;
   CoordSaldaturaPP11[9].Y2 := L#-197398;
   CoordSaldaturaPP11[10].X1 := L#-56162;
   CoordSaldaturaPP11[10].Y1 := L#-210332;
   CoordSaldaturaPP11[10].X2 := L#-56200;
   CoordSaldaturaPP11[10].Y2 := L#-210331;
   CoordSaldaturaPP11[11].X1 := L#-40981;
   CoordSaldaturaPP11[11].Y1 := L#-215911;
   CoordSaldaturaPP11[11].X2 := L#-40587;
   CoordSaldaturaPP11[11].Y2 := L#-215681;
   CoordinateCam_PP1[1].X := L#7915;
   CoordinateCam_PP1[1].Y := L#-68282;
   NumeroSaldaturePP1 := 10;
   TimeWeldingPP1[1].Tempo := S5T#1S;
   TimeWeldingPP1[2].Tempo := S5T#2S;
   TimeWeldingPP1[3].Tempo := S5T#1S;
   TimeWeldingPP1[4].Tempo := S5T#1S;
   TimeWeldingPP1[5].Tempo := S5T#1S;
   TimeWeldingPP1[6].Tempo := S5T#1S;
   TimeWeldingPP1[7].Tempo := S5T#1S;
   TimeWeldingPP1[8].Tempo := S5T#1S;
   TimeWeldingPP1[9].Tempo := S5T#1S;
   TimeWeldingPP1[10].Tempo := S5T#1S;
   TimeWeldingPP1[11].Tempo := S5T#1S;
   TimeWeldingPP1[12].Tempo := S5T#1S;
   TimeWeldingPP1[13].Tempo := S5T#1S;
   TimeWeldingPP1[14].Tempo := S5T#1S;
   TimeWeldingPP1[15].Tempo := S5T#1S;
   TimeWeldingPP1[16].Tempo := S5T#1S;
   TimeWeldingPP1[17].Tempo := S5T#1S;
   TimeWeldingPP1[18].Tempo := S5T#1S;
   TimeWeldingPP1[19].Tempo := S5T#1S;
   TimeWeldingPP1[20].Tempo := S5T#1S;
   TimeWeldingPP2[1].Tempo := S5T#1S;
   TimeWeldingPP2[2].Tempo := S5T#1S;
   TimeWeldingPP2[3].Tempo := S5T#1S;
   TimeWeldingPP2[4].Tempo := S5T#1S;
   TimeWeldingPP2[5].Tempo := S5T#1S;
   TimeWeldingPP2[6].Tempo := S5T#1S;
   TimeWeldingPP2[7].Tempo := S5T#1S;
   TimeWeldingPP2[8].Tempo := S5T#1S;
   TimeWeldingPP2[9].Tempo := S5T#1S;
   TimeWeldingPP2[10].Tempo := S5T#1S;
   TimeWeldingPP2[11].Tempo := S5T#1S;
   TimeWeldingPP2[12].Tempo := S5T#1S;
   TimeWeldingPP2[13].Tempo := S5T#1S;
   TimeWeldingPP2[14].Tempo := S5T#1S;
   TimeWeldingPP2[15].Tempo := S5T#1S;
   TimeWeldingPP2[16].Tempo := S5T#1S;
   TimeWeldingPP2[17].Tempo := S5T#1S;
   TimeWeldingPP2[18].Tempo := S5T#1S;
   TimeWeldingPP2[19].Tempo := S5T#1S;
   TimeWeldingPP2[20].Tempo := S5T#1S;
   TimeWeldingPP3[1].Tempo := S5T#1S;
   TimeWeldingPP3[2].Tempo := S5T#1S;
   TimeWeldingPP3[3].Tempo := S5T#1S;
   TimeWeldingPP3[4].Tempo := S5T#1S;
   TimeWeldingPP3[5].Tempo := S5T#1S;
   TimeWeldingPP3[6].Tempo := S5T#1S;
   TimeWeldingPP3[7].Tempo := S5T#1S;
   TimeWeldingPP3[8].Tempo := S5T#1S;
   TimeWeldingPP3[9].Tempo := S5T#1S;
   TimeWeldingPP3[10].Tempo := S5T#1S;
   TimeWeldingPP3[11].Tempo := S5T#1S;
   TimeWeldingPP3[12].Tempo := S5T#1S;
   TimeWeldingPP3[13].Tempo := S5T#1S;
   TimeWeldingPP3[14].Tempo := S5T#1S;
   TimeWeldingPP3[15].Tempo := S5T#1S;
   TimeWeldingPP3[16].Tempo := S5T#1S;
   TimeWeldingPP3[17].Tempo := S5T#1S;
   TimeWeldingPP3[18].Tempo := S5T#1S;
   TimeWeldingPP3[19].Tempo := S5T#1S;
   TimeWeldingPP3[20].Tempo := S5T#1S;
   TimeWeldingPP4[1].Tempo := S5T#1S;
   TimeWeldingPP4[2].Tempo := S5T#1S;
   TimeWeldingPP4[3].Tempo := S5T#1S;
   TimeWeldingPP4[4].Tempo := S5T#1S;
   TimeWeldingPP4[5].Tempo := S5T#1S;
   TimeWeldingPP4[6].Tempo := S5T#1S;
   TimeWeldingPP4[7].Tempo := S5T#1S;
   TimeWeldingPP4[8].Tempo := S5T#1S;
   TimeWeldingPP4[9].Tempo := S5T#1S;
   TimeWeldingPP4[10].Tempo := S5T#1S;
   TimeWeldingPP4[11].Tempo := S5T#1S;
   TimeWeldingPP4[12].Tempo := S5T#1S;
   TimeWeldingPP4[13].Tempo := S5T#1S;
   TimeWeldingPP4[14].Tempo := S5T#1S;
   TimeWeldingPP4[15].Tempo := S5T#1S;
   TimeWeldingPP4[16].Tempo := S5T#1S;
   TimeWeldingPP4[17].Tempo := S5T#1S;
   TimeWeldingPP4[18].Tempo := S5T#1S;
   TimeWeldingPP4[19].Tempo := S5T#1S;
   TimeWeldingPP4[20].Tempo := S5T#1S;
   TimeWeldingPP5[1].Tempo := S5T#1S;
   TimeWeldingPP5[2].Tempo := S5T#1S;
   TimeWeldingPP5[3].Tempo := S5T#1S;
   TimeWeldingPP5[4].Tempo := S5T#1S;
   TimeWeldingPP5[5].Tempo := S5T#1S;
   TimeWeldingPP5[6].Tempo := S5T#1S;
   TimeWeldingPP5[7].Tempo := S5T#1S;
   TimeWeldingPP5[8].Tempo := S5T#1S;
   TimeWeldingPP5[9].Tempo := S5T#1S;
   TimeWeldingPP5[10].Tempo := S5T#1S;
   TimeWeldingPP5[11].Tempo := S5T#1S;
   TimeWeldingPP5[12].Tempo := S5T#1S;
   TimeWeldingPP5[13].Tempo := S5T#1S;
   TimeWeldingPP5[14].Tempo := S5T#1S;
   TimeWeldingPP5[15].Tempo := S5T#1S;
   TimeWeldingPP5[16].Tempo := S5T#1S;
   TimeWeldingPP5[17].Tempo := S5T#1S;
   TimeWeldingPP5[18].Tempo := S5T#1S;
   TimeWeldingPP5[19].Tempo := S5T#1S;
   TimeWeldingPP5[20].Tempo := S5T#1S;
   TimeWeldingPP6[1].Tempo := S5T#1S;
   TimeWeldingPP6[2].Tempo := S5T#1S;
   TimeWeldingPP6[3].Tempo := S5T#1S;
   TimeWeldingPP6[4].Tempo := S5T#1S;
   TimeWeldingPP6[5].Tempo := S5T#1S;
   TimeWeldingPP6[6].Tempo := S5T#1S;
   TimeWeldingPP6[7].Tempo := S5T#1S;
   TimeWeldingPP6[8].Tempo := S5T#1S;
   TimeWeldingPP6[9].Tempo := S5T#1S;
   TimeWeldingPP6[10].Tempo := S5T#1S;
   TimeWeldingPP6[11].Tempo := S5T#1S;
   TimeWeldingPP6[12].Tempo := S5T#1S;
   TimeWeldingPP6[13].Tempo := S5T#1S;
   TimeWeldingPP6[14].Tempo := S5T#1S;
   TimeWeldingPP6[15].Tempo := S5T#1S;
   TimeWeldingPP6[16].Tempo := S5T#1S;
   TimeWeldingPP6[17].Tempo := S5T#1S;
   TimeWeldingPP6[18].Tempo := S5T#1S;
   TimeWeldingPP6[19].Tempo := S5T#1S;
   TimeWeldingPP6[20].Tempo := S5T#1S;
   TimeWeldingPP7[1].Tempo := S5T#1S;
   TimeWeldingPP7[2].Tempo := S5T#1S;
   TimeWeldingPP7[3].Tempo := S5T#1S;
   TimeWeldingPP7[4].Tempo := S5T#1S;
   TimeWeldingPP7[5].Tempo := S5T#1S;
   TimeWeldingPP7[6].Tempo := S5T#1S;
   TimeWeldingPP7[7].Tempo := S5T#1S;
   TimeWeldingPP7[8].Tempo := S5T#1S;
   TimeWeldingPP7[9].Tempo := S5T#1S;
   TimeWeldingPP7[10].Tempo := S5T#1S;
   TimeWeldingPP7[11].Tempo := S5T#1S;
   TimeWeldingPP7[12].Tempo := S5T#1S;
   TimeWeldingPP7[13].Tempo := S5T#1S;
   TimeWeldingPP7[14].Tempo := S5T#1S;
   TimeWeldingPP7[15].Tempo := S5T#1S;
   TimeWeldingPP7[16].Tempo := S5T#1S;
   TimeWeldingPP7[17].Tempo := S5T#1S;
   TimeWeldingPP7[18].Tempo := S5T#1S;
   TimeWeldingPP7[19].Tempo := S5T#1S;
   TimeWeldingPP7[20].Tempo := S5T#1S;
   TimeWeldingPP8[1].Tempo := S5T#1S;
   TimeWeldingPP8[2].Tempo := S5T#1S;
   TimeWeldingPP8[3].Tempo := S5T#1S;
   TimeWeldingPP8[4].Tempo := S5T#1S;
   TimeWeldingPP8[5].Tempo := S5T#1S;
   TimeWeldingPP8[6].Tempo := S5T#1S;
   TimeWeldingPP8[7].Tempo := S5T#1S;
   TimeWeldingPP8[8].Tempo := S5T#1S;
   TimeWeldingPP8[9].Tempo := S5T#1S;
   TimeWeldingPP8[10].Tempo := S5T#1S;
   TimeWeldingPP8[11].Tempo := S5T#1S;
   TimeWeldingPP8[12].Tempo := S5T#1S;
   TimeWeldingPP8[13].Tempo := S5T#1S;
   TimeWeldingPP8[14].Tempo := S5T#1S;
   TimeWeldingPP8[15].Tempo := S5T#1S;
   TimeWeldingPP8[16].Tempo := S5T#1S;
   TimeWeldingPP8[17].Tempo := S5T#1S;
   TimeWeldingPP8[18].Tempo := S5T#1S;
   TimeWeldingPP8[19].Tempo := S5T#1S;
   TimeWeldingPP8[20].Tempo := S5T#1S;
   TimeWeldingPP9[1].Tempo := S5T#1S;
   TimeWeldingPP9[2].Tempo := S5T#1S;
   TimeWeldingPP9[3].Tempo := S5T#1S;
   TimeWeldingPP9[4].Tempo := S5T#1S;
   TimeWeldingPP9[5].Tempo := S5T#1S;
   TimeWeldingPP9[6].Tempo := S5T#1S;
   TimeWeldingPP9[7].Tempo := S5T#1S;
   TimeWeldingPP9[8].Tempo := S5T#1S;
   TimeWeldingPP9[9].Tempo := S5T#1S;
   TimeWeldingPP9[10].Tempo := S5T#1S;
   TimeWeldingPP9[11].Tempo := S5T#1S;
   TimeWeldingPP9[12].Tempo := S5T#1S;
   TimeWeldingPP9[13].Tempo := S5T#1S;
   TimeWeldingPP9[14].Tempo := S5T#1S;
   TimeWeldingPP9[15].Tempo := S5T#1S;
   TimeWeldingPP9[16].Tempo := S5T#1S;
   TimeWeldingPP9[17].Tempo := S5T#1S;
   TimeWeldingPP9[18].Tempo := S5T#1S;
   TimeWeldingPP9[19].Tempo := S5T#1S;
   TimeWeldingPP9[20].Tempo := S5T#1S;
   TimeWeldingPP10[1].Tempo := S5T#1S;
   TimeWeldingPP10[2].Tempo := S5T#1S;
   TimeWeldingPP10[3].Tempo := S5T#1S;
   TimeWeldingPP10[4].Tempo := S5T#1S;
   TimeWeldingPP10[5].Tempo := S5T#1S;
   TimeWeldingPP10[6].Tempo := S5T#1S;
   TimeWeldingPP10[7].Tempo := S5T#1S;
   TimeWeldingPP10[8].Tempo := S5T#1S;
   TimeWeldingPP10[9].Tempo := S5T#1S;
   TimeWeldingPP10[10].Tempo := S5T#1S;
   TimeWeldingPP10[11].Tempo := S5T#1S;
   TimeWeldingPP10[12].Tempo := S5T#1S;
   TimeWeldingPP10[13].Tempo := S5T#1S;
   TimeWeldingPP10[14].Tempo := S5T#1S;
   TimeWeldingPP10[15].Tempo := S5T#1S;
   TimeWeldingPP10[16].Tempo := S5T#1S;
   TimeWeldingPP10[17].Tempo := S5T#1S;
   TimeWeldingPP10[18].Tempo := S5T#1S;
   TimeWeldingPP10[19].Tempo := S5T#1S;
   TimeWeldingPP10[20].Tempo := S5T#1S;
   TimeWeldingPP11[1].Tempo := S5T#1S700MS;
   TimeWeldingPP11[2].Tempo := S5T#1S;
   TimeWeldingPP11[3].Tempo := S5T#1S;
   TimeWeldingPP11[4].Tempo := S5T#1S;
   TimeWeldingPP11[5].Tempo := S5T#1S;
   TimeWeldingPP11[6].Tempo := S5T#1S;
   TimeWeldingPP11[7].Tempo := S5T#1S;
   TimeWeldingPP11[8].Tempo := S5T#1S;
   TimeWeldingPP11[9].Tempo := S5T#1S;
   TimeWeldingPP11[10].Tempo := S5T#1S;
   TimeWeldingPP11[11].Tempo := S5T#1S;
   TimeWeldingPP11[12].Tempo := S5T#1S;
   TimeWeldingPP11[13].Tempo := S5T#1S;
   TimeWeldingPP11[14].Tempo := S5T#1S;
   TimeWeldingPP11[15].Tempo := S5T#1S;
   TimeWeldingPP11[16].Tempo := S5T#1S;
   TimeWeldingPP11[17].Tempo := S5T#1S;
   TimeWeldingPP11[18].Tempo := S5T#1S;
   TimeWeldingPP11[19].Tempo := S5T#1S;
   TimeWeldingPP11[20].Tempo := S5T#1S;
   TimeWeldingPP12[1].Tempo := S5T#1S;
   TimeWeldingPP12[2].Tempo := S5T#1S;
   TimeWeldingPP12[3].Tempo := S5T#1S;
   TimeWeldingPP12[4].Tempo := S5T#1S;
   TimeWeldingPP12[5].Tempo := S5T#1S;
   TimeWeldingPP12[6].Tempo := S5T#1S;
   TimeWeldingPP12[7].Tempo := S5T#1S;
   TimeWeldingPP12[8].Tempo := S5T#1S;
   TimeWeldingPP12[9].Tempo := S5T#1S;
   TimeWeldingPP12[10].Tempo := S5T#1S;
   TimeWeldingPP12[11].Tempo := S5T#1S;
   TimeWeldingPP12[12].Tempo := S5T#1S;
   TimeWeldingPP12[13].Tempo := S5T#1S;
   TimeWeldingPP12[14].Tempo := S5T#1S;
   TimeWeldingPP12[15].Tempo := S5T#1S;
   TimeWeldingPP12[16].Tempo := S5T#1S;
   TimeWeldingPP12[17].Tempo := S5T#1S;
   TimeWeldingPP12[18].Tempo := S5T#1S;
   TimeWeldingPP12[19].Tempo := S5T#1S;
   TimeWeldingPP12[20].Tempo := S5T#1S;
   TimeWeldingPP13[1].Tempo := S5T#1S;
   TimeWeldingPP13[2].Tempo := S5T#1S;
   TimeWeldingPP13[3].Tempo := S5T#1S;
   TimeWeldingPP13[4].Tempo := S5T#1S;
   TimeWeldingPP13[5].Tempo := S5T#1S;
   TimeWeldingPP13[6].Tempo := S5T#1S;
   TimeWeldingPP13[7].Tempo := S5T#1S;
   TimeWeldingPP13[8].Tempo := S5T#1S;
   TimeWeldingPP13[9].Tempo := S5T#1S;
   TimeWeldingPP13[10].Tempo := S5T#1S;
   TimeWeldingPP13[11].Tempo := S5T#1S;
   TimeWeldingPP13[12].Tempo := S5T#1S;
   TimeWeldingPP13[13].Tempo := S5T#1S;
   TimeWeldingPP13[14].Tempo := S5T#1S;
   TimeWeldingPP13[15].Tempo := S5T#1S;
   TimeWeldingPP13[16].Tempo := S5T#1S;
   TimeWeldingPP13[17].Tempo := S5T#1S;
   TimeWeldingPP13[18].Tempo := S5T#1S;
   TimeWeldingPP13[19].Tempo := S5T#1S;
   TimeWeldingPP13[20].Tempo := S5T#1S;
   TimeWeldingPP14[1].Tempo := S5T#1S;
   TimeWeldingPP14[2].Tempo := S5T#1S;
   TimeWeldingPP14[3].Tempo := S5T#1S;
   TimeWeldingPP14[4].Tempo := S5T#1S;
   TimeWeldingPP14[5].Tempo := S5T#1S;
   TimeWeldingPP14[6].Tempo := S5T#1S;
   TimeWeldingPP14[7].Tempo := S5T#1S;
   TimeWeldingPP14[8].Tempo := S5T#1S;
   TimeWeldingPP14[9].Tempo := S5T#1S;
   TimeWeldingPP14[10].Tempo := S5T#1S;
   TimeWeldingPP14[11].Tempo := S5T#1S;
   TimeWeldingPP14[12].Tempo := S5T#1S;
   TimeWeldingPP14[13].Tempo := S5T#1S;
   TimeWeldingPP14[14].Tempo := S5T#1S;
   TimeWeldingPP14[15].Tempo := S5T#1S;
   TimeWeldingPP14[16].Tempo := S5T#1S;
   TimeWeldingPP14[17].Tempo := S5T#1S;
   TimeWeldingPP14[18].Tempo := S5T#1S;
   TimeWeldingPP14[19].Tempo := S5T#1S;
   TimeWeldingPP14[20].Tempo := S5T#1S;
   TimeWeldingPP15[1].Tempo := S5T#1S;
   TimeWeldingPP15[2].Tempo := S5T#1S;
   TimeWeldingPP15[3].Tempo := S5T#1S;
   TimeWeldingPP15[4].Tempo := S5T#1S;
   TimeWeldingPP15[5].Tempo := S5T#1S;
   TimeWeldingPP15[6].Tempo := S5T#1S;
   TimeWeldingPP15[7].Tempo := S5T#1S;
   TimeWeldingPP15[8].Tempo := S5T#1S;
   TimeWeldingPP15[9].Tempo := S5T#1S;
   TimeWeldingPP15[10].Tempo := S5T#1S;
   TimeWeldingPP15[11].Tempo := S5T#1S;
   TimeWeldingPP15[12].Tempo := S5T#1S;
   TimeWeldingPP15[13].Tempo := S5T#1S;
   TimeWeldingPP15[14].Tempo := S5T#1S;
   TimeWeldingPP15[15].Tempo := S5T#1S;
   TimeWeldingPP15[16].Tempo := S5T#1S;
   TimeWeldingPP15[17].Tempo := S5T#1S;
   TimeWeldingPP15[18].Tempo := S5T#1S;
   TimeWeldingPP15[19].Tempo := S5T#1S;
   TimeWeldingPP15[20].Tempo := S5T#1S;
   TimeWeldingPP16[1].Tempo := S5T#1S;
   TimeWeldingPP16[2].Tempo := S5T#1S;
   TimeWeldingPP16[3].Tempo := S5T#1S;
   TimeWeldingPP16[4].Tempo := S5T#1S;
   TimeWeldingPP16[5].Tempo := S5T#1S;
   TimeWeldingPP16[6].Tempo := S5T#1S;
   TimeWeldingPP16[7].Tempo := S5T#1S;
   TimeWeldingPP16[8].Tempo := S5T#1S;
   TimeWeldingPP16[9].Tempo := S5T#1S;
   TimeWeldingPP16[10].Tempo := S5T#1S;
   TimeWeldingPP16[11].Tempo := S5T#1S;
   TimeWeldingPP16[12].Tempo := S5T#1S;
   TimeWeldingPP16[13].Tempo := S5T#1S;
   TimeWeldingPP16[14].Tempo := S5T#1S;
   TimeWeldingPP16[15].Tempo := S5T#1S;
   TimeWeldingPP16[16].Tempo := S5T#1S;
   TimeWeldingPP16[17].Tempo := S5T#1S;
   TimeWeldingPP16[18].Tempo := S5T#1S;
   TimeWeldingPP16[19].Tempo := S5T#1S;
   TimeWeldingPP16[20].Tempo := S5T#1S;
   TimeWeldingPP17[1].Tempo := S5T#1S;
   TimeWeldingPP17[2].Tempo := S5T#1S;
   TimeWeldingPP17[3].Tempo := S5T#1S;
   TimeWeldingPP17[4].Tempo := S5T#1S;
   TimeWeldingPP17[5].Tempo := S5T#1S;
   TimeWeldingPP17[6].Tempo := S5T#1S;
   TimeWeldingPP17[7].Tempo := S5T#1S;
   TimeWeldingPP17[8].Tempo := S5T#1S;
   TimeWeldingPP17[9].Tempo := S5T#1S;
   TimeWeldingPP17[10].Tempo := S5T#1S;
   TimeWeldingPP17[11].Tempo := S5T#1S;
   TimeWeldingPP17[12].Tempo := S5T#1S;
   TimeWeldingPP17[13].Tempo := S5T#1S;
   TimeWeldingPP17[14].Tempo := S5T#1S;
   TimeWeldingPP17[15].Tempo := S5T#1S;
   TimeWeldingPP17[16].Tempo := S5T#1S;
   TimeWeldingPP17[17].Tempo := S5T#1S;
   TimeWeldingPP17[18].Tempo := S5T#1S;
   TimeWeldingPP17[19].Tempo := S5T#1S;
   TimeWeldingPP17[20].Tempo := S5T#1S;
   TimeWeldingPP18[1].Tempo := S5T#1S;
   TimeWeldingPP18[2].Tempo := S5T#1S;
   TimeWeldingPP18[3].Tempo := S5T#1S;
   TimeWeldingPP18[4].Tempo := S5T#1S;
   TimeWeldingPP18[5].Tempo := S5T#1S;
   TimeWeldingPP18[6].Tempo := S5T#1S;
   TimeWeldingPP18[7].Tempo := S5T#1S;
   TimeWeldingPP18[8].Tempo := S5T#1S;
   TimeWeldingPP18[9].Tempo := S5T#1S;
   TimeWeldingPP18[10].Tempo := S5T#1S;
   TimeWeldingPP18[11].Tempo := S5T#1S;
   TimeWeldingPP18[12].Tempo := S5T#1S;
   TimeWeldingPP18[13].Tempo := S5T#1S;
   TimeWeldingPP18[14].Tempo := S5T#1S;
   TimeWeldingPP18[15].Tempo := S5T#1S;
   TimeWeldingPP18[16].Tempo := S5T#1S;
   TimeWeldingPP18[17].Tempo := S5T#1S;
   TimeWeldingPP18[18].Tempo := S5T#1S;
   TimeWeldingPP18[19].Tempo := S5T#1S;
   TimeWeldingPP18[20].Tempo := S5T#1S;
   TimeWeldingPP19[1].Tempo := S5T#1S;
   TimeWeldingPP19[2].Tempo := S5T#1S;
   TimeWeldingPP19[3].Tempo := S5T#1S;
   TimeWeldingPP19[4].Tempo := S5T#1S;
   TimeWeldingPP19[5].Tempo := S5T#1S;
   TimeWeldingPP19[6].Tempo := S5T#1S;
   TimeWeldingPP19[7].Tempo := S5T#1S;
   TimeWeldingPP19[8].Tempo := S5T#1S;
   TimeWeldingPP19[9].Tempo := S5T#1S;
   TimeWeldingPP19[10].Tempo := S5T#1S;
   TimeWeldingPP19[11].Tempo := S5T#1S;
   TimeWeldingPP19[12].Tempo := S5T#1S;
   TimeWeldingPP19[13].Tempo := S5T#1S;
   TimeWeldingPP19[14].Tempo := S5T#1S;
   TimeWeldingPP19[15].Tempo := S5T#1S;
   TimeWeldingPP19[16].Tempo := S5T#1S;
   TimeWeldingPP19[17].Tempo := S5T#1S;
   TimeWeldingPP19[18].Tempo := S5T#1S;
   TimeWeldingPP19[19].Tempo := S5T#1S;
   TimeWeldingPP19[20].Tempo := S5T#1S;
   TimeWeldingPP20[1].Tempo := S5T#1S;
   TimeWeldingPP20[2].Tempo := S5T#1S;
   TimeWeldingPP20[3].Tempo := S5T#1S;
   TimeWeldingPP20[4].Tempo := S5T#1S;
   TimeWeldingPP20[5].Tempo := S5T#1S;
   TimeWeldingPP20[6].Tempo := S5T#1S;
   TimeWeldingPP20[7].Tempo := S5T#1S;
   TimeWeldingPP20[8].Tempo := S5T#1S;
   TimeWeldingPP20[9].Tempo := S5T#1S;
   TimeWeldingPP20[10].Tempo := S5T#1S;
   TimeWeldingPP20[11].Tempo := S5T#1S;
   TimeWeldingPP20[12].Tempo := S5T#1S;
   TimeWeldingPP20[13].Tempo := S5T#1S;
   TimeWeldingPP20[14].Tempo := S5T#1S;
   TimeWeldingPP20[15].Tempo := S5T#1S;
   TimeWeldingPP20[16].Tempo := S5T#1S;
   TimeWeldingPP20[17].Tempo := S5T#1S;
   TimeWeldingPP20[18].Tempo := S5T#1S;
   TimeWeldingPP20[19].Tempo := S5T#1S;
   TimeWeldingPP20[20].Tempo := S5T#1S;
END_DATA_BLOCK

DATA_BLOCK "DB180"	// DB 180
VERSION : 0.1
"FB24 - Gestione Mov Assi"
BEGIN
END_DATA_BLOCK

DATA_BLOCK "DB181"	// DB 181
VERSION : 0.1
"FB24 - Gestione Mov Assi"
BEGIN
END_DATA_BLOCK

ORGANIZATION_BLOCK "MAIN PROGRAM"	// OB 1
TITLE = "Main Program Sweep (Cycle)"
VERSION : 0.1
VAR_TEMP
  OB1_EV_CLASS : BYTE ;	//Bits 0-3 = 1 (Coming event), Bits 4-7 = 1 (Event class 1)
  OB1_SCAN_1 : BYTE ;	//1 (Cold restart scan 1 of OB 1), 3 (Scan 2-n of OB 1)
  OB1_PRIORITY : BYTE ;	//Priority of OB Execution
  OB1_OB_NUMBR : BYTE ;	//1 (Organization block 1, OB1)
  OB1_RESERVED_1 : BYTE ;	//Reserved for system
  OB1_RESERVED_2 : BYTE ;	//Reserved for system
  OB1_PREV_CYCLE : INT ;	//Cycle time of previous OB1 scan (milliseconds)
  OB1_MIN_CYCLE : INT ;	//Minimum cycle time of OB1 (milliseconds)
  OB1_MAX_CYCLE : INT ;	//Maximum cycle time of OB1 (milliseconds)
  OB1_DATE_TIME : DATE_AND_TIME ;	//Date and time OB1 started
END_VAR
BEGIN
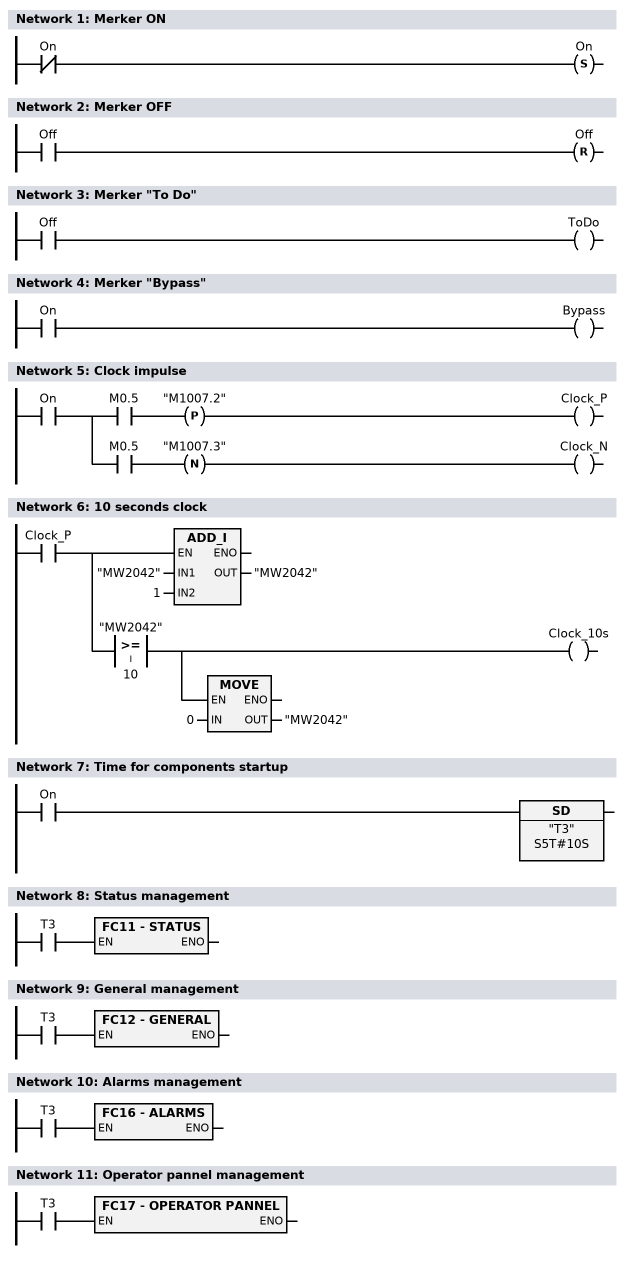
NETWORK
TITLE = Merker ON
      AN    "On";
      S     "On";
NETWORK
TITLE = Merker OFF
      A     "Off";
      R     "Off";
NETWORK
TITLE = Merker "To Do"
      A     "Off";
      =     "ToDo";
NETWORK
TITLE = Merker "Bypass"
      A     "On";
      =     "Bypass";
NETWORK
TITLE = Clock impulse
      A     "On";
      =     L 20.0;
      A     L 20.0;
      A     "M0.5";
      FP    "M1007.2";
      =     "Clock_P";
      A     L 20.0;
      A     "M0.5";
      FN    "M1007.3";
      =     "Clock_N";
NETWORK
TITLE = 10 seconds clock
      A     "Clock_P";
      =     L 20.0;
      A     L 20.0;
      JNB   _001;
      L     "MW2042";
      L     1;
      +I;
      T     "MW2042";
_001: NOP   0;
      A     L 20.0;
      A(;
      L     "MW2042";
      L     10;
      >=I;
      );
      =     L 20.1;
      A     L 20.1;
      BLD   102;
      =     "Clock_10s";
      A     L 20.1;
      JNB   _002;
      L     0;
      T     "MW2042";
_002: NOP   0;
NETWORK
TITLE = Time for components startup
      A     "On";
      L     S5T#10S;
      SD    "T3";
NETWORK
TITLE = Status management
      A     "T3";
      JNB   _003;
      CALL  "FC11 - STATUS";
_003: NOP   0;
NETWORK
TITLE = General management
      A     "T3";
      JNB   _004;
      CALL  "FC12 - GENERAL";
_004: NOP   0;
NETWORK
TITLE = Alarms management
      A     "T3";
      JNB   _005;
      CALL  "FC16 - ALARMS";
_005: NOP   0;
NETWORK
TITLE = Operator pannel management
      A     "T3";
      JNB   _006;
      CALL  "FC17 - OPERATOR PANNEL";
_006: NOP   0;
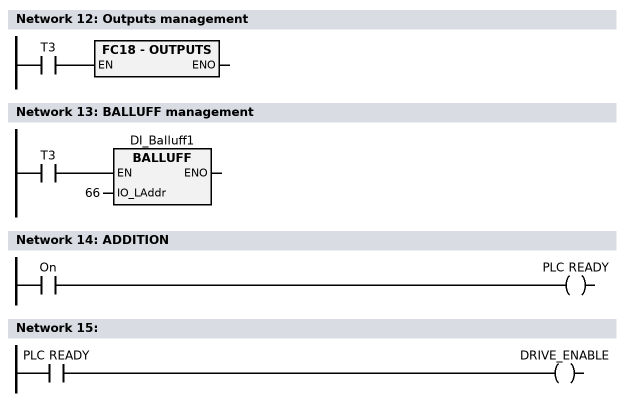
NETWORK
TITLE = Outputs management
      A     "T3";
      JNB   _007;
      CALL  "FC18 - OUTPUTS";
_007: NOP   0;
NETWORK
TITLE = BALLUFF management
      A     "T3";
      JNB   _008;
      CALL  "BALLUFF" , "DI_Balluff1" (
           IO_LAddr                 := 66);
_008: NOP   0;
NETWORK
TITLE = ADDITION
      A     "On";
      =     "PLC READY";
NETWORK
TITLE =
      A     "PLC READY";
      =     "DRIVE_ENABLE";
END_ORGANIZATION_BLOCK

ORGANIZATION_BLOCK "I/O_FLT1"	// OB 82
TITLE = "I/O Point Fault"
VERSION : 1.0
VAR_TEMP
  OB82_EV_CLASS : BYTE ;	// 16#39, Event class 3, entering event state, internal fault event
  OB82_FLT_ID : BYTE ;	// 16#XX, Fault identification code
  OB82_PRIORITY : BYTE ;	// 26/28 (Priority of 1 is lowest)
  OB82_OB_NUMBR : BYTE ;	// 82 (Organization block 82, OB82)
  OB82_RESERVED_1 : BYTE ;	// Reserved for system
  OB82_IO_FLAG : BYTE ;	// Input (01010100), Output (01010101)
  OB82_MDL_ADDR : INT ;	// Base address of module with fault
  OB82_MDL_DEFECT : BOOL ;	// Module defective
  OB82_INT_FAULT : BOOL ;	// Internal fault
  OB82_EXT_FAULT : BOOL ;	// External fault
  OB82_PNT_INFO : BOOL ;	// Point information
  OB82_EXT_VOLTAGE : BOOL ;	// External voltage low
  OB82_FLD_CONNCTR : BOOL ;	// Field wiring connector missing
  OB82_NO_CONFIG : BOOL ;	// Module has no configuration data
  OB82_CONFIG_ERR : BOOL ;	// Module has configuration error
  OB82_MDL_TYPE : BYTE ;	// Type of module
  OB82_SUB_NDL_ERR : BOOL ;	// Sub-Module is missing or has error
  OB82_COMM_FAULT : BOOL ;	// Communication fault
  OB82_MDL_STOP : BOOL ;	// Module is stopped
  OB82_WTCH_DOG_FLT : BOOL ;	// Watch dog timer stopped module
  OB82_INT_PS_FLT : BOOL ;	// Internal power supply fault
  OB82_PRIM_BATT_FLT : BOOL ;	// Primary battery is faulty
  OB82_BCKUP_BATT_FLT : BOOL ;	// Backup battery is faulty
  OB82_RESERVED_2 : BOOL ;	// Reserved for system
  OB82_RACK_FLT : BOOL ;	// Rack fault, only for bus interface module
  OB82_PROC_FLT : BOOL ;	// Processor fault
  OB82_EPROM_FLT : BOOL ;	// EPROM fault
  OB82_RAM_FLT : BOOL ;	// RAM fault
  OB82_ADU_FLT : BOOL ;	// ADC fault
  OB82_FUSE_FLT : BOOL ;	// Fuse fault
  OB82_HW_INTR_FLT : BOOL ;	// Hardware interrupt input faulty
  OB82_RESERVED_3 : BOOL ;	// Reserved for system
  OB82_DATE_TIME : DATE_AND_TIME ;	// Date and time OB82 started
END_VAR
BEGIN
NETWORK
TITLE =
END_ORGANIZATION_BLOCK

ORGANIZATION_BLOCK "RACK_FLT"	// OB 86
TITLE = "Loss Of Rack Fault"
VERSION : 0.1
VAR_TEMP
  OB86_EV_CLASS : BYTE ;	//16#38/39 Event class 3
  OB86_FLT_ID : BYTE ;	//16#C1/C4/C5, Fault identifcation code
  OB86_PRIORITY : BYTE ;	//Priority of OB Execution
  OB86_OB_NUMBR : BYTE ;	//86 (Organization block 86, OB86)
  OB86_RESERVED_1 : BYTE ;	//Reserved for system
  OB86_RESERVED_2 : BYTE ;	//Reserved for system
  OB86_MDL_ADDR : WORD ;	//Base address of IM module in rack with fault
  OB86_RACKS_FLTD : ARRAY  [0 .. 31 ] OF BOOL ;	//Racks in fault
  OB86_DATE_TIME : DATE_AND_TIME ;	//Date and time OB86 started
END_VAR
BEGIN
NETWORK
TITLE =
END_ORGANIZATION_BLOCK

ORGANIZATION_BLOCK "COMPLETE RESTART"	// OB 100
TITLE = "Complete Restart"
VERSION : 0.1
VAR_TEMP
  OB100_EV_CLASS : BYTE ;	//16#13, Event class 1, Entering event state, Event logged in diagnostic buffer
  OB100_STRTUP : BYTE ;	//16#81/82/83/84 Method of startup
  OB100_PRIORITY : BYTE ;	//Priority of OB Execution
  OB100_OB_NUMBR : BYTE ;	//100 (Organization block 100, OB100)
  OB100_RESERVED_1 : BYTE ;	//Reserved for system
  OB100_RESERVED_2 : BYTE ;	//Reserved for system
  OB100_STOP : WORD ;	//Event that caused CPU to stop (16#4xxx)
  OB100_STRT_INFO : DWORD ;	//Information on how system started
  OB100_DATE_TIME : DATE_AND_TIME ;	//Date and time OB100 started
END_VAR
BEGIN
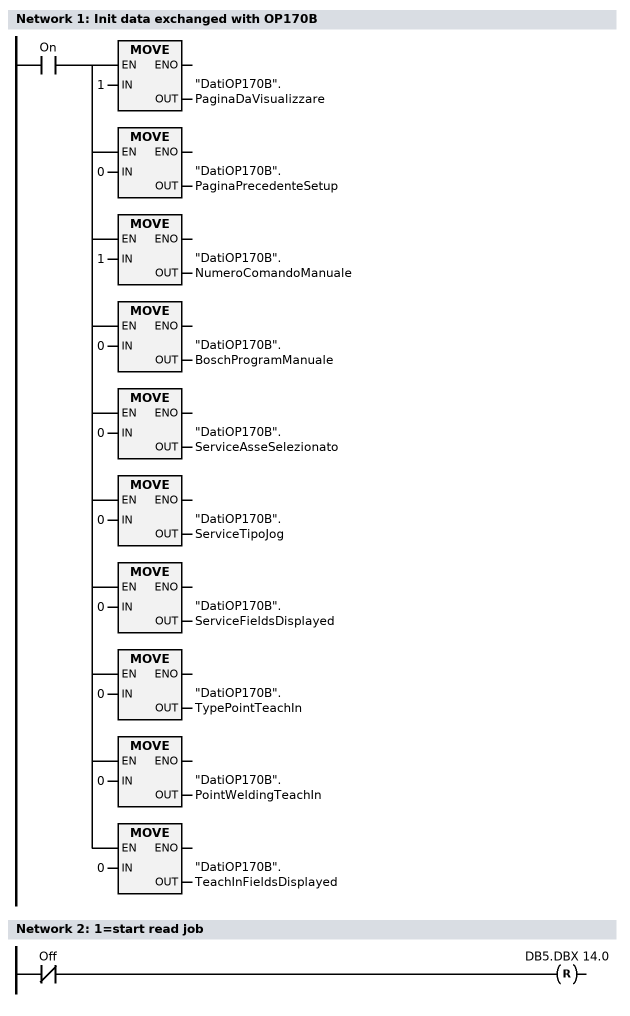
NETWORK
TITLE = Init data exchanged with OP170B
      A     "On";
      =     L 20.0;
      A     L 20.0;
      JNB   _001;
      L     1;
      T     "DatiOP170B".PaginaDaVisualizzare;
_001: NOP   0;
      A     L 20.0;
      JNB   _002;
      L     0;
      T     "DatiOP170B".PaginaPrecedenteSetup;
_002: NOP   0;
      A     L 20.0;
      JNB   _003;
      L     1;
      T     "DatiOP170B".NumeroComandoManuale;
_003: NOP   0;
      A     L 20.0;
      JNB   _004;
      L     0;
      T     "DatiOP170B".BoschProgramManuale;
_004: NOP   0;
      A     L 20.0;
      JNB   _005;
      L     0;
      T     "DatiOP170B".ServiceAsseSelezionato;
_005: NOP   0;
      A     L 20.0;
      JNB   _006;
      L     0;
      T     "DatiOP170B".ServiceTipoJog;
_006: NOP   0;
      A     L 20.0;
      JNB   _007;
      L     0;
      T     "DatiOP170B".ServiceFieldsDisplayed;
_007: NOP   0;
      A     L 20.0;
      JNB   _008;
      L     0;
      T     "DatiOP170B".TypePointTeachIn;
_008: NOP   0;
      A     L 20.0;
      JNB   _009;
      L     0;
      T     "DatiOP170B".PointWeldingTeachIn;
_009: NOP   0;
      A     L 20.0;
      JNB   _00a;
      L     0;
      T     "DatiOP170B".TeachInFieldsDisplayed;
_00a: NOP   0;
NETWORK
TITLE = 1=start read job
      AN    "Off";
      R     DB5.DBX 14.0;
END_ORGANIZATION_BLOCK

ORGANIZATION_BLOCK "MOD_ERR"	// OB 122
TITLE = "Module Access Error"
VERSION : 0.1
VAR_TEMP
  OB122_EV_CLASS : BYTE ;	//16#29, Event class 2, Entering event state, Internal fault event
  OB122_SW_FLT : BYTE ;	//16#XX Software error code
  OB122_PRIORITY : BYTE ;	//Priority of OB Execution
  OB122_OB_NUMBR : BYTE ;	//122 (Organization block 122, OB122)
  OB122_BLK_TYPE : BYTE ;	//16#88/8C/8E Type of block fault occured in
  OB122_MEM_AREA : BYTE ;	//Memory area where access error occured
  OB122_MEM_ADDR : WORD ;	//Memory address where access error occured
  OB122_BLK_NUM : WORD ;	//Block number in which error occured
  OB122_PRG_ADDR : WORD ;	//Program address where error occured
  OB122_DATE_TIME : DATE_AND_TIME ;	//Date and time OB1 started
END_VAR
BEGIN
NETWORK
TITLE =
END_ORGANIZATION_BLOCK

SYMBOL_TABLE
"DI_Balluff1"	DB 5	FB 20	// DB Instance of FB20
"DatiOP170B"	DB 7	DB 7	// PLC<->OP170B interface
"Timer"	DB 20	DB 20
"DBWork"	DB 21	DB 21
"coordinate"	DB 22	DB 22
"DB180"	DB 180	FB 24	// DB instance FB24 AsseY
"DB181"	DB 181	FB 24	// DB instance FB24 AsseX
"Asse_611U"	FB 16	FB 16	// Axis 611U management
"BALLUFF"	FB 20	FB 20	// BALLUFF Reader/Writer management
"FB24 - Gestione Mov Assi"	FB 24	FB 24	// GESTIONE ASSI STAZIONE
"NormalizzazioneAnalogico"	FC 7	FC 7	// Normalization of a analog value
"FC11 - STATUS"	FC 11	FC 11	// Sensors and proximity state
"FC12 - GENERAL"	FC 12	FC 12	// General management
"FC13 - MANUAL"	FC 13	FC 13	// Manual commands
"FC14 - AUTOMATIC"	FC 14	FC 14	// Automatic cycle management
"FC16 - ALARMS"	FC 16	FC 16	// Alarms management
"FC17 - OPERATOR PANNEL"	FC 17	FC 17	// Operator pannel management
"FC18 - OUTPUTS"	FC 18	FC 18	// Outputs management
"FC19 - REPOSITIONING"	FC 19	FC 19	// Repositioning management
"FC50 - TEACH-IN"	FC 50	FC 50
"FC51 - TYPE TOOL"	FC 51	FC 51
"FC52 - SYSTEM VISION"	FC 52	FC 52
"FC53 - REWORK"	FC 53	FC 53
"FC81 - GEST AXIS"	FC 81	FC 81	// Management axis
"FC117 - ERROR TOOL"	FC 117	FC 117
"TimeOut"	FC 800	FC 800	// Management TimeOut movimenti
"MAIN PROGRAM"	OB 1	OB 1	// Main Program
"I/O_FLT1"	OB 82	OB 82	// I/O Point Fault 1
"RACK_FLT"	OB 86	OB 86	// Loss of Rack Fault
"COMPLETE RESTART"	OB 100	OB 100	// Complete Restart
"MOD_ERR"	OB 122	OB 122	// Module Access Error
"TON"	SFB 4	SFB 4	// Generate an On Delay
"READ_CLK"	SFC 1	SFC 1	// Read System Clock
"DPRD_DAT"	SFC 14	SFC 14	// Read Consistent Data of a Standard DP Slave
"DPWR_DAT"	SFC 15	SFC 15	// Write Consistent Data to a Standard DP Slave
"BLKMOV"	SFC 20	SFC 20	// Copy Variables
"FILL"	SFC 21	SFC 21	// Initialize a Memory Area
"CREAT_DB"	SFC 22	SFC 22	// Create Data Block
"DIS_AIRT"	SFC 41	SFC 41	// Delay the Higher Priority Interrupts and Asynchronous Errors
"EN_AIRT"	SFC 42	SFC 42	// Enable Higher Priority Interrupts and Asynchronous Errors
"STP"	SFC 46	SFC 46	// Change the CPU to STOP
"LGC_GADR"	SFC 49	SFC 49	// Query the Module Slot Belonging to a Logical Address
"RDSYSST"	SFC 51	SFC 51	// Read a System Status List or Partial List
"WR_REC"	SFC 58	SFC 58	// Write Data Record
"RD_REC"	SFC 59	SFC 59	// Read a Data Record
"VAT_1"	VAT 1	
"Coordinate_saldatura"	VAT 2	
"I/O System Vision"	VAT 3	
"Saldatrice"	VAT 4	
"VAT_12"	VAT 5	
"VAT_17"	VAT 6	
"VAT_Balluff"	VAT 7	
"DB22_SaldaturaSilv"	VAT 8	
"DB22_Sald_PP1"	VAT 9	
"VAT_Daniele"	VAT 10	
"VAT_Point"	VAT 11	
"ASSE_P"	VAT 12	
"DB22_Sald_PP3"	VAT 13	
"VAT_Point 16"	VAT 14	
"VAT_PUNTI_AVV"	VAT 15	
"DB22_Sald_PP16"	VAT 16	
"VAT_PUNTI_AVV_2"	VAT 17	
"Tipo portapezzo"	VAT 18	
"VAT_tool check"	VAT 19	
END_SYMBOL_TABLE

FUNCTION_BLOCK "Asse_611U"	// FB 16
TITLE = Axis 611U management
VERSION : 0.1
VAR_INPUT
  IO_LAddr : INT ;	//Logic address of the inputs/outputs
END_VAR
VAR
  In_Profibus : STRUCT 	//Inputs from 611U (via Profibus)
   PKW : STRUCT 	//Parameter area of the Profibus telegram
    PKE : WORD ;
    IND : WORD ;
    PWE : DINT ;
   END_STRUCT ;
   PZD : STRUCT 	//Process data area of the Profibus telegram
    ZSW1 : STRUCT 	//Status word 1
     Bit8 : BOOL ;	//Following error (0=following error outside the window error)
     Bit9 : BOOL ;	//DP control requested (1=DP master is requested to accept control)
     Bit10 : BOOL ;	//Reference position reached (1=end of traversing block reached)
     Bit11 : BOOL ;	//Reference point set (1=axis is referenced)
     Bit12 : BOOL ;	//Setpoint acknowledge (1=the traversing task is processed)
     Bit13 : BOOL ;	//Drive stationery (1=drive is not in movement)
     Bit14 : BOOL ;	//External block change selected
     Bit15 : BOOL ;	//Request passive referencing
     Bit0 : BOOL ;	//Ready to switch-on (1=ready to power-up)
     Bit1 : BOOL ;	//Ready or no fault (1=drive ready or no fault present)
     Bit2 : BOOL ;	//Controller enable (1=speed controller active and setpoint can be accepted)
     Bit3 : BOOL ;	//Fault present (1=fault present)
     Bit4 : BOOL ;	//No OFF2 (1=OFF2 not present)
     Bit5 : BOOL ;	//No OFF3 (1=OFF3 not present)
     Bit6 : BOOL ;	//Switch-on inhibit (1=power-on inhibit)
     Bit7 : BOOL ;	//Alarm present (1=alarm present)
    END_STRUCT ;
    AktSatz : STRUCT 	//Actual block status word
     Bit8 : BOOL ;	//Reserved
     Bit9 : BOOL ;	//Reserved
     Bit10 : BOOL ;	//Reserved
     Bit11 : BOOL ;	//Reserved
     Bit12 : BOOL ;	//Reserved
     Bit13 : BOOL ;	//Reserved
     Bit14 : BOOL ;	//Reserved
     Bit15 : BOOL ;	//MDI Active
     Bit0 : BOOL ;	//Bit 0 block selected
     Bit1 : BOOL ;	//Bit 1 block selected
     Bit2 : BOOL ;	//Bit 2 block selected
     Bit3 : BOOL ;	//Bit 3 block selected
     Bit4 : BOOL ;	//Bit 4 block selected
     Bit5 : BOOL ;	//Bit 5 block selected
     Bit6 : BOOL ;	//Reserved
     Bit7 : BOOL ;	//Reserved
    END_STRUCT ;
    PosZsw : STRUCT 	//Position status word
     Bit8 : BOOL ;	//Cam switching signal 1
     Bit9 : BOOL ;	//Cam switching signal 2
     Bit10 : BOOL ;	//Direct output 1 via the traversing block
     Bit11 : BOOL ;	//Direct output 2 via the traversing block
     Bit12 : BOOL ;	//Fixed endstop reached
     Bit13 : BOOL ;	//Fixed endstop clamping torque reached
     Bit14 : BOOL ;	//Traverse to fixed endstop active
     Bit15 : BOOL ;	//Teach-In executed
     Bit0 : BOOL ;	//Tracking mode active (1=tracking mode active)
     Bit1 : BOOL ;	//Velocity limiting (1=velocity is limited)
     Bit2 : BOOL ;	//Setpoint stationary (1=axis stationary on the setpoint side)
     Bit3 : BOOL ;	//In synchronism (1=slave drive is synchronized with the master drive)
     Bit4 : BOOL ;	//Axis moves forwards
     Bit5 : BOOL ;	//Axis moves backwards
     Bit6 : BOOL ;	//Minus software limit switch actuated
     Bit7 : BOOL ;	//Plus software limit switch actuated
    END_STRUCT ;
    ZSW2 : STRUCT 	//Status word 2
     Bit8 : BOOL ;	//Suppress fault 608 active
     Bit9 : BOOL ;	//n.u. (used only in the n-set mode)
     Bit10 : BOOL ;	//n.u. (used only in the n-set mode)
     Bit11 : BOOL ;	//n.u. (used only in the n-set mode)
     Bit12 : BOOL ;	//Slave sign-of-life
     Bit13 : BOOL ;	//Slave sign-of-life
     Bit14 : BOOL ;	//Slave sign-of-life
     Bit15 : BOOL ;	//Slave sign-of-life
     Bit0 : BOOL ;	//Bit 0 parameter set
     Bit1 : BOOL ;	//Bit 1 parameter set
     Bit2 : BOOL ;	//Bit 2 parameter set
     Bit3 : BOOL ;	//First speed setpoint filter inactive
     Bit4 : BOOL ;	//Rump-function generator inactive
     Bit5 : BOOL ;	//Open holding brake
     Bit6 : BOOL ;	//Integrator inhibit
     Bit7 : BOOL ;	//Parking axis selected
    END_STRUCT ;
    XretrP : DINT ;	//Actual position value
    DIG_IN : STRUCT 	//Digital inputs status
     Bit8 : BOOL ;
     Bit9 : BOOL ;
     Bit10 : BOOL ;
     Bit11 : BOOL ;
     Bit12 : BOOL ;
     Bit13 : BOOL ;
     Bit14 : BOOL ;
     Bit15 : BOOL ;
     Bit0 : BOOL ;	//Axis on home cam
     Bit1 : BOOL ;	//Axis on minus extra-corse limit switch
     Bit2 : BOOL ;	//Axis on plus extra-corse limit switch
     Bit3 : BOOL ;
     Bit4 : BOOL ;
     Bit5 : BOOL ;
     Bit6 : BOOL ;
     Bit7 : BOOL ;
    END_STRUCT ;
   END_STRUCT ;
  END_STRUCT ;
  Out_Profibus : STRUCT 	//Outputs to 611U (via Profibus)
   PKW : STRUCT 	//Parameter area of the Profibus telegram
    PKE : WORD ;
    IND : WORD ;
    PWE : DINT ;
   END_STRUCT ;
   PZD : STRUCT 	//Process data area of the Profibus telegram
    STW1 : STRUCT 	//Control word 1
     Bit8 : BOOL ;	//JOG1 (1=the drive traverse with the speed in P0108)
     Bit9 : BOOL ;	//JOG2 (1=the drive traverse with the speed in P0109)
     Bit10 : BOOL ;	//Control requested (Should be set 1 when ZSW1.9=1)
     Bit11 : BOOL ;	//Stop referencing (1=start the referencing point approach)
     Bit12 : BOOL ;	//Opening the holding brake for test purposes
     Bit13 : BOOL ;	//External block change (With a edge the external block changing is initiated)
     Bit14 : BOOL ;	//Reserved
     Bit15 : BOOL ;	//Request passive referencing
     Bit0 : BOOL ;	//OFF1 (1=enable)
     Bit1 : BOOL ;	//OFF2 (1=enable)
     Bit2 : BOOL ;	//OFF3 (1=enable)
     Bit3 : BOOL ;	//Pulse inhibit (0=the motor stop for inertia)
     Bit4 : BOOL ;	//Reject travel task (0=stop the motor and delete the distance to go)
     Bit5 : BOOL ;	//Intermediate stop (0=stop the motor but the process is continued with 0/1 edge)
     Bit6 : BOOL ;	//Activate travel task (With a edge the traversing block selected is started)
     Bit7 : BOOL ;	//Reset the fault memory (1=Reset the fault memory)
    END_STRUCT ;
    SatzAnw : STRUCT 	//Block selection control word
     Bit8 : BOOL ;	//Reserved
     Bit9 : BOOL ;	//Reserved
     Bit10 : BOOL ;	//Reserved
     Bit11 : BOOL ;	//Reserved
     Bit12 : BOOL ;	//Reserved
     Bit13 : BOOL ;	//Reserved
     Bit14 : BOOL ;	//Reserved
     Bit15 : BOOL ;	//Activate MDI
     Bit0 : BOOL ;	//Bit 0 block selection
     Bit1 : BOOL ;	//Bit 1 block selection
     Bit2 : BOOL ;	//Bit 2 block selection
     Bit3 : BOOL ;	//Bit 3 block selection
     Bit4 : BOOL ;	//Bit 4 block selection
     Bit5 : BOOL ;	//Bit 5 block selection
     Bit6 : BOOL ;	//Reserved
     Bit7 : BOOL ;	//Reserved
    END_STRUCT ;
    PosStw : STRUCT 	//Position control word
     Bit8 : BOOL ;	//Reserved
     Bit9 : BOOL ;	//Reserved
     Bit10 : BOOL ;	//Reserved
     Bit11 : BOOL ;	//Reserved
     Bit12 : BOOL ;	//Reserved
     Bit13 : BOOL ;	//Reserved
     Bit14 : BOOL ;	//Reserved
     Bit15 : BOOL ;	//Reserved
     Bit0 : BOOL ;	//Tracking operation (1=select tracking operation)
     Bit1 : BOOL ;	//Set reference point (0/1 edge=P0160 is assigned as actual value)
     Bit2 : BOOL ;	//Reference cams (1=the axis is located at reference cam)
     Bit3 : BOOL ;	//Fixed endstop (1=fixed endstop reached)
     Bit4 : BOOL ;	//Activate the coupling (0/1 edge=activate coupling set via P0410)
     BIt5 : BOOL ;	//Incremental jogging (1=jog in velocity and increments)
     Bit6 : BOOL ;	//Activate Teach-In (0/1=Activate Teach-In; 1/0=Reset Teach-In)
     Bit7 : BOOL ;	//Invert the angular encoder input
    END_STRUCT ;
    STW2 : STRUCT 	//Control word 2
     Bit8 : BOOL ;	//Suppress fault 608
     Bit9 : BOOL ;	//n.u. (used only in the n-set mode)
     Bit10 : BOOL ;	//n.u. (used only in the n-set mode)
     Bit11 : BOOL ;	//n.u. (used only in the n-set mode)
     Bit12 : BOOL ;	//Master sign-of-life
     Bit13 : BOOL ;	//Master sign-of-life
     Bit14 : BOOL ;	//Master sign-of-life
     Bit15 : BOOL ;	//Master sign-of-life
     Bit0 : BOOL ;	//Bit 0 parameter set changeover
     Bit1 : BOOL ;	//Bit 1 parameter set changeover
     Bit2 : BOOL ;	//Bit 2 parameter set changeover
     Bit3 : BOOL ;	//First speed setpoint filter disabled
     Bit4 : BOOL ;	//Rump-function generator enabled
     Bit5 : BOOL ;	//Reserved
     Bit6 : BOOL ;	//Integrator inhibit
     Bit7 : BOOL ;	//Select parking axis
    END_STRUCT ;
    Over : INT ;	//Percentage value for the velocity override
   END_STRUCT ;
  END_STRUCT ;
  Enable : BOOL ;	//Enable the drive
  Reset_Alarms : BOOL ;	//Reset the alarms
  Reset_Axis : BOOL ;	//Stop all the movements
  Start_Inc : BOOL ;	//Start incremental movement
  Start_Abs : BOOL ;	//Start absolute movement
  Start_Rep : BOOL ;	//Start repositioning movement
  Start_Ref : BOOL ;	//Start referencing movement
  Stop : BOOL ;	//Intermediate stop movement
  Jog_Forward : BOOL ;	//Jog forward command
  Jog_Backward : BOOL ;	//Jog backward command
  STAT58 : BOOL ;	//Reserved
  STAT57 : BOOL ;	//Reserved
  STAT56 : BOOL ;	//Reserved
  STAT55 : BOOL ;	//Reserved
  STAT54 : BOOL ;	//Reserved
  STAT53 : BOOL ;	//Reserved
  Step1_Inc : BOOL ;	//Step 1 for incremental movement management
  Step2_Inc : BOOL ;	//Step 2 for incremental movement management
  Step1_Abs : BOOL ;	//Step 1 for absolute movement management
  Step2_Abs : BOOL ;	//Step 2 for absolute movement management
  STAT36 : BOOL ;	//Reserved
  STAT35 : BOOL ;	//Reserved
  STAT34 : BOOL ;	//Reserved
  STAT33 : BOOL ;	//Reserved
  InZeroPosition : BOOL ;	//Axis in "zero" position
  AxisStationery : BOOL ;	//Axis stationery
  DriveOK : BOOL ;	//Drive OK
  BrakeOpen : BOOL ;	//Open holding brake request
  AxisOnHWHomeCam : BOOL ;	//Axis on hardware home cam
  AxisOnHWSwitchN : BOOL ;	//Axis on minus hardware extra-corse limit switch
  AxisOnHWSwitchP : BOOL ;	//Axis on plus hardware extra-corse limit switch
  AxisOnSWSwitchN : BOOL ;	//Axis on minus software extra-corse limit switch
  AxisOnSWSwitchP : BOOL ;	//Axis on plus software extra-corse limit switch
  STAT69 : BOOL ;	//Reserved
  STAT67 : BOOL ;	//Reserved
  STAT66 : BOOL ;	//Reserved
  STAT65 : BOOL ;	//Reserved
  STAT64 : BOOL ;	//Reserved
  STAT63 : BOOL ;	//Reserved
  STAT70 : BOOL ;	//Reserved
  Aux1 : BOOL ;	//Auxiliary for edge management
  Aux2 : BOOL ;	//Auxiliary for edge management
  Aux3 : BOOL ;	//Auxiliary for edge management
  Aux4 : BOOL ;	//Auxiliary for edge management
  Aux5 : BOOL ;	//Auxiliary for edge management
  Aux6 : BOOL ;	//Auxiliary for edge management
  Aux7 : BOOL ;	//Auxiliary for edge management
  Aux8 : BOOL ;	//Auxiliary for edge management
  Target_Inc : DINT ;	//Target for the incremental movement
  Target_Abs : DINT ;	//Target for the absolute movement
  DistanceToGo_Abs : DINT ;	//Difference between actual and new position
  Override : INT ;	//Percentage value for the velocity override
  ActualPosition : DINT ;	//Actual position value
END_VAR
VAR_TEMP
  tempAR1 : DWORD ;
  tempAR2 : DWORD ;
  tempSRC : ANY ;
  tempDST : ANY ;
  tempDWORD_1 : DWORD ;
  tempWORD_1 : WORD ;
  tempINT : INT ;
  tempDWORD_2 : DWORD ;
END_VAR
BEGIN
NETWORK
TITLE = Mapping of the inputs
      L     #IO_LAddr;
      SLD   3;
      T     #tempDWORD_1;
      L     P##In_Profibus;
      T     #tempDWORD_2;
      L     11;
NXT1: T     #tempINT;
      L     PIW [#tempDWORD_1];
      T     DIW [#tempDWORD_2];
      L     #tempDWORD_1;
      L     P#2.0;
      +D;
      T     #tempDWORD_1;
      L     #tempDWORD_2;
      L     P#2.0;
      +D;
      T     #tempDWORD_2;
      L     #tempINT;
      LOOP  NXT1;
NETWORK
TITLE = Status
//Axis stationery
      A     #In_Profibus.PZD.ZSW1.Bit13;
      AN    #In_Profibus.PZD.ZSW1.Bit12;
      =     #AxisStationery;
//Drive OK
      A     #In_Profibus.PZD.ZSW1.Bit0;
      A     #In_Profibus.PZD.ZSW1.Bit1;
      A     #In_Profibus.PZD.ZSW1.Bit2;
      AN    #In_Profibus.PZD.ZSW1.Bit3;
      A     #In_Profibus.PZD.ZSW1.Bit4;
      A     #In_Profibus.PZD.ZSW1.Bit5;
      A     #In_Profibus.PZD.ZSW1.Bit8;
      =     #DriveOK;
//Open holding brake request
      A     #In_Profibus.PZD.ZSW2.Bit5;
      =     #BrakeOpen;
//Axis on hardware home cam
      A     #In_Profibus.PZD.DIG_IN.Bit0;
      =     #AxisOnHWHomeCam;
//Axis on hardware minus extra-course limit switch
      A     #In_Profibus.PZD.DIG_IN.Bit1;
      =     #AxisOnHWSwitchN;
//Axis on hardware plus extra-course limit switch
      A     #In_Profibus.PZD.DIG_IN.Bit2;
      =     #AxisOnHWSwitchP;
//Axis on software minus extra-course limit switch
      A     #In_Profibus.PZD.PosZsw.Bit6;
      =     #AxisOnSWSwitchN;
//Axis on software plus extra-course limit switch
      A     #In_Profibus.PZD.PosZsw.Bit7;
      =     #AxisOnSWSwitchP;
//Actual position value
      L     #In_Profibus.PZD.XretrP;
      T     #ActualPosition;
NETWORK
TITLE = Commands
//Enable the drive
      A     #Enable;
      =     #Out_Profibus.PZD.STW1.Bit0;
      =     #Out_Profibus.PZD.STW1.Bit1;
      =     #Out_Profibus.PZD.STW1.Bit2;
      A     M 1.1;
      =     #Out_Profibus.PZD.STW1.Bit3;
//Erase all the movements
      O     #Reset_Axis;
      O     #In_Profibus.PZD.ZSW1.Bit3;
      ON    #In_Profibus.PZD.ZSW1.Bit8;
      R     #Start_Inc;
      R     #Step1_Inc;
      R     #Step2_Inc;
      R     #Start_Abs;
      R     #Step1_Abs;
      R     #Step2_Abs;
      R     #Start_Rep;
      R     #Start_Ref;
      R     #Out_Profibus.PZD.STW1.Bit11;
      R     #Out_Profibus.PZD.STW1.Bit6;
//Stop the axis and erase the distance to go
      AN    #Reset_Axis;
      =     #Out_Profibus.PZD.STW1.Bit4;
//Intermediate stop the axis (the movement continued with a 0/1 edge)
      AN    #Stop;
      =     #Out_Profibus.PZD.STW1.Bit5;
//Reset alarms
      A     #Reset_Alarms;
      =     #Out_Profibus.PZD.STW1.Bit7;
//Control request (611U<->PLC communication)
      A     #In_Profibus.PZD.ZSW1.Bit9;
      =     #Out_Profibus.PZD.STW1.Bit10;
//Velocity override
      L     #Override;
      T     #Out_Profibus.PZD.Over;
NETWORK
TITLE = Movement in incremental mode
//Reset the incremental movement if the axis is the distance to go is minus then 0,05mm
      A     #Start_Inc;
      A(;
      L     #Target_Inc;
      L     50;
      <D;
      );
      A(;
      L     #Target_Inc;
      L     -50;
      >D;
      );
      R     #Start_Inc;
//Select the travel block (Block number 2=000010)
      A     #Start_Inc;
      R     #Out_Profibus.PZD.SatzAnw.Bit0;
      S     #Out_Profibus.PZD.SatzAnw.Bit1;
      R     #Out_Profibus.PZD.SatzAnw.Bit2;
      R     #Out_Profibus.PZD.SatzAnw.Bit3;
      R     #Out_Profibus.PZD.SatzAnw.Bit4;
      R     #Out_Profibus.PZD.SatzAnw.Bit5;
//Load the new position of the travel block
      A     #Start_Inc;
      AN    #Step1_Inc;
      AN    #Step2_Inc;
      S     #Step1_Inc;
      JCN   L001;
      L     #Target_Inc;
      T     #Out_Profibus.PKW.PWE;
      L     W#16#8051;
      T     #Out_Profibus.PKW.PKE;
      L     2;
      T     #Out_Profibus.PKW.IND;
L001: NOP   0;
//Check if the 611U received the change
      A     #Start_Inc;
      A     #Step1_Inc;
      AN    #Step2_Inc;
      A(;
      L     #Out_Profibus.PKW.PWE;
      L     #In_Profibus.PKW.PWE;
      ==D;
      );
      A(;
      L     W#16#5051;
      L     #In_Profibus.PKW.PKE;
      ==I;
      );
      A(;
      L     #Out_Profibus.PKW.IND;
      L     #In_Profibus.PKW.IND;
      ==I;
      );
      S     #Step2_Inc;
//Start travel task
      A     #Start_Inc;
      A     #Step1_Inc;
      A     #Step2_Inc;
      A(;
      L     #Target_Inc;
      L     #In_Profibus.PKW.PWE;
      ==D;
      );
//UN    #In_Profibus.PZD.AktSatz.Bit0
//U     #In_Profibus.PZD.AktSatz.Bit1
//UN    #In_Profibus.PZD.AktSatz.Bit2
//UN    #In_Profibus.PZD.AktSatz.Bit3
//UN    #In_Profibus.PZD.AktSatz.Bit4
//UN    #In_Profibus.PZD.AktSatz.Bit5
      AN    #Out_Profibus.PZD.STW1.Bit6;
      S     #Out_Profibus.PZD.STW1.Bit6;
      JCN   L002;
      L     0;
      T     #Out_Profibus.PKW.PKE;
      T     #Out_Profibus.PKW.IND;
      T     #Out_Profibus.PKW.PWE;
L002: NOP   0;
//End incremental movement
      A     #In_Profibus.PZD.ZSW1.Bit10;
      FP    #Aux1;
      A     #Start_Inc;
      A     #Step1_Inc;
      A     #Step2_Inc;
      A     #Out_Profibus.PZD.STW1.Bit6;
      R     #Out_Profibus.PZD.STW1.Bit6;
      R     #Start_Inc;
      R     #Step1_Inc;
      R     #Step2_Inc;
NETWORK
TITLE = Movement in absolute mode
//Movement not necessary if the axis is just in position  
      A     #Start_Abs;
      AN    #Step1_Abs;
      AN    #Step2_Abs;
      JCN   L004;
//Calculate the difference between the actual position and new position
      L     #Target_Abs;
      L     #In_Profibus.PZD.XretrP;
      -D;
      T     #DistanceToGo_Abs;
      L     0;
      <D;
      JCN   L003;
      L     #DistanceToGo_Abs;
      NEGD;
      T     #DistanceToGo_Abs;
L003: NOP   0;
      A(;
      L     #DistanceToGo_Abs;
      L     99;
      <=D;
      );
      R     #Start_Abs;
L004: NOP   0;
//Select the travel block (Block number 0=000000)
      A     #Start_Abs;
      R     #Out_Profibus.PZD.SatzAnw.Bit0;
      R     #Out_Profibus.PZD.SatzAnw.Bit1;
      R     #Out_Profibus.PZD.SatzAnw.Bit2;
      R     #Out_Profibus.PZD.SatzAnw.Bit3;
      R     #Out_Profibus.PZD.SatzAnw.Bit4;
      R     #Out_Profibus.PZD.SatzAnw.Bit5;
//Load the new position of the travel block
      A     #Start_Abs;
      AN    #Step1_Abs;
      AN    #Step2_Abs;
      S     #Step1_Abs;
      JCN   L005;
      L     #Target_Abs;
      T     #Out_Profibus.PKW.PWE;
      L     W#16#8051;
      T     #Out_Profibus.PKW.PKE;
      L     0;
      T     #Out_Profibus.PKW.IND;
L005: NOP   0;
//Check if the 611U received the change
      A     #Start_Abs;
      A     #Step1_Abs;
      AN    #Step2_Abs;
      A(;
      L     #Out_Profibus.PKW.PWE;
      L     #In_Profibus.PKW.PWE;
      ==D;
      );
      A(;
      L     W#16#5051;
      L     #In_Profibus.PKW.PKE;
      ==I;
      );
      A(;
      L     #Out_Profibus.PKW.IND;
      L     #In_Profibus.PKW.IND;
      ==I;
      );
      S     #Step2_Abs;
//Start travel task
      A     #Start_Abs;
      A     #Step1_Abs;
      A     #Step2_Abs;
      A(;
      L     #Target_Abs;
      L     #In_Profibus.PKW.PWE;
      ==D;
      );
      AN    #In_Profibus.PZD.AktSatz.Bit0;
      AN    #In_Profibus.PZD.AktSatz.Bit1;
      AN    #In_Profibus.PZD.AktSatz.Bit2;
      AN    #In_Profibus.PZD.AktSatz.Bit3;
      AN    #In_Profibus.PZD.AktSatz.Bit4;
      AN    #In_Profibus.PZD.AktSatz.Bit5;
      AN    #Out_Profibus.PZD.STW1.Bit6;
      S     #Out_Profibus.PZD.STW1.Bit6;
      JCN   L006;
      L     0;
      T     #Out_Profibus.PKW.PKE;
      T     #Out_Profibus.PKW.IND;
      T     #Out_Profibus.PKW.PWE;
L006: NOP   0;
//End absolute movement
      A     #In_Profibus.PZD.ZSW1.Bit10;
      FP    #Aux2;
      A     #Start_Abs;
      A     #Step1_Abs;
      A     #Step2_Abs;
      A     #Out_Profibus.PZD.STW1.Bit6;
      R     #Out_Profibus.PZD.STW1.Bit6;
      R     #Start_Abs;
      R     #Step1_Abs;
      R     #Step2_Abs;
NETWORK
TITLE = Repositioning management
//Movement not necessary if the axis is just in position  
      A     #Start_Rep;
      FP    #Aux3;
      A     #InZeroPosition;
      R     #Start_Rep;
//Select the travel block (Block number 1=000001)
      A     #Start_Rep;
      S     #Out_Profibus.PZD.SatzAnw.Bit0;
      R     #Out_Profibus.PZD.SatzAnw.Bit1;
      R     #Out_Profibus.PZD.SatzAnw.Bit2;
      R     #Out_Profibus.PZD.SatzAnw.Bit3;
      R     #Out_Profibus.PZD.SatzAnw.Bit4;
      R     #Out_Profibus.PZD.SatzAnw.Bit5;
//Start travel task
      A     #Start_Rep;
      A     #In_Profibus.PZD.AktSatz.Bit0;
      AN    #In_Profibus.PZD.AktSatz.Bit1;
      AN    #In_Profibus.PZD.AktSatz.Bit2;
      AN    #In_Profibus.PZD.AktSatz.Bit3;
      AN    #In_Profibus.PZD.AktSatz.Bit4;
      AN    #In_Profibus.PZD.AktSatz.Bit5;
      AN    #Out_Profibus.PZD.STW1.Bit6;
      S     #Out_Profibus.PZD.STW1.Bit6;
//End repositioning
      A     #In_Profibus.PZD.ZSW1.Bit10;
      FP    #Aux4;
      A     #Start_Rep;
      A     #Out_Profibus.PZD.STW1.Bit6;
      R     #Out_Profibus.PZD.STW1.Bit6;
      R     #Start_Rep;
NETWORK
TITLE = Jog management
//Jog forward
      A     #Jog_Forward;
      A     #In_Profibus.PZD.ZSW1.Bit11;
      AN    #In_Profibus.PZD.PosZsw.Bit7;
      =     #Out_Profibus.PZD.STW1.Bit9;
//Jog backward
      A     #Jog_Backward;
      A     #In_Profibus.PZD.ZSW1.Bit11;
      AN    #In_Profibus.PZD.PosZsw.Bit6;
      =     #Out_Profibus.PZD.STW1.Bit8;
NETWORK
TITLE = Referencing management
//Start the referencing point approach
      A     #Start_Ref;
      FP    #Aux5;
      S     #Out_Profibus.PZD.STW1.Bit11;
//End of referencing point approch
      A     #In_Profibus.PZD.ZSW1.Bit11;
      FP    #Aux6;
      R     #Out_Profibus.PZD.STW1.Bit11;
      R     #Start_Ref;
NETWORK
TITLE = Mapping of the outputs
      L     #IO_LAddr;
      SLD   3;
      T     #tempDWORD_1;
      L     P##Out_Profibus;
      T     #tempDWORD_2;
      L     9;
NXT3: T     #tempINT;
      L     DIW [#tempDWORD_2];
      T     PQW [#tempDWORD_1];
      L     #tempDWORD_1;
      L     P#2.0;
      +D;
      T     #tempDWORD_1;
      L     #tempDWORD_2;
      L     P#2.0;
      +D;
      T     #tempDWORD_2;
      L     #tempINT;
      LOOP  NXT3;
END_FUNCTION_BLOCK

FUNCTION_BLOCK "BALLUFF"	// FB 20
TITLE = BALLUFF Reader/Writer management
VERSION : 0.1
VAR_INPUT
  IO_LAddr : INT ;
END_VAR
VAR
  InputBuffer : STRUCT
   CP : BOOL ;	//Codetag present
   AA : BOOL ;	//Command started
   AE : BOOL ;	//Command finished without error
   AF : BOOL ;	//Command finished with error
   KN : BOOL ;	//Header number
   TO : BOOL ;	//Toggle-bit Out
   HF : BOOL ;	//Head error
   BB : BOOL ;	//Ready
   ErrorCode : BYTE ;
   Data1 : BYTE ;
   Data2 : BYTE ;
   Data3 : BYTE ;
   Data4 : BYTE ;
  END_STRUCT ;
  OutputBuffer : STRUCT
   AV : BOOL ;	//Command
   Reserved1 : BOOL ;
   GR : BOOL ;	//Ground state
   Reserved2 : BOOL ;
   HD : BOOL ;	//Head direct
   Reserved3 : BOOL ;
   TI : BOOL ;	//Toggle-bit in
   CT : BOOL ;	//Codetag type
   Command : BYTE ;
   StartAddress_L : BYTE ;
   StartAddress_H : BYTE ;
   NoBytes_L : BYTE ;
   NoBytes_H : BYTE ;
  END_STRUCT ;
  Testa1 : STRUCT
   Lettura_Start : BOOL ;	//1=start read job
   Lettura_OK : BOOL ;	//1=read job ended without error
   Lettura_NOK : BOOL ;	//1=read job ended with error
   Lettura_Step1 : BOOL ;	//Aux for read job cycle
   Lettura_Step2 : BOOL ;	//Aux for read job cycle
   Lettura_Step3 : BOOL ;	//Aux for read job cycle
   Lettura_Step4 : BOOL ;	//Aux for read job cycle
   Lettura_Step5 : BOOL ;	//Aux for read job cycle
   Scrittura_Start : BOOL ;	//1=start write job
   Scrittura_OK : BOOL ;	//1=write job ended without error
   Scrittura_NOK : BOOL ;	//1=write job ended with error
   Scrittura_Step1 : BOOL ;	//Aux for write job cycle
   Scrittura_Step2 : BOOL ;	//Aux for write job cycle
   Scrittura_Step3 : BOOL ;	//Aux for write job cycle
   Scrittura_Step4 : BOOL ;	//Aux for write job cycle
   Scrittura_Step5 : BOOL ;	//Aux for write job cycle
   ValoreLetto : BYTE ;	//Data readed
   ValoreDaScrivere : BYTE ;	//Data to write
   Seconds : BYTE ;	//Number of seconds of activity
  END_STRUCT ;
  Testa2 : STRUCT
   Lettura_Start : BOOL ;	//1=start read job
   Lettura_OK : BOOL ;	//1=read job ended without error
   Lettura_NOK : BOOL ;	//1=read job ended with error
   Lettura_Step1 : BOOL ;	//Aux for read job cycle
   Lettura_Step2 : BOOL ;	//Aux for read job cycle
   Lettura_Step3 : BOOL ;	//Aux for read job cycle
   Lettura_Step4 : BOOL ;	//Aux for read job cycle
   Lettura_Step5 : BOOL ;	//Aux for read job cycle
   Scrittura_Start : BOOL ;	//1=start write job
   Scrittura_OK : BOOL ;	//1=write job ended without error
   Scrittura_NOK : BOOL ;	//1=write job ended with error
   Scrittura_Step1 : BOOL ;	//Aux for write job cycle
   Scrittura_Step2 : BOOL ;	//Aux for write job cycle
   Scrittura_Step3 : BOOL ;	//Aux for write job cycle
   Scrittura_Step4 : BOOL ;	//Aux for write job cycle
   Scrittura_Step5 : BOOL ;	//Aux for write job cycle
   ValoreLetto : BYTE ;	//Data readed
   ValoreDaScrivere : BYTE ;	//Data to write
   Seconds : BYTE ;	//Number of seconds of activity
  END_STRUCT ;
END_VAR
VAR_TEMP
  tempAR1 : DWORD ;
  tempAR2 : DWORD ;
  tempSRC : ANY ;
  tempDST : ANY ;
  tempDWORD_1 : DWORD ;
  tempWORD_1 : WORD ;
  tempINT : INT ;
  tempBYTE1 : BYTE ;
  tempBYTE2 : BYTE ;
END_VAR
BEGIN
NETWORK
TITLE = Mapping of the inputs
//Save registry value
      TAR1  #tempAR1;
      TAR2  #tempAR2;
//Creation of a pointer to the source area
      LAR1  P##tempSRC;	//Load initial address of source pointer in AR1
      L     B#16#10;	//Load the ID for the ANY type
      T     LB [AR1,P#0.0];
      L     B#16#2;	//2=type of data is BYTE
      T     LB [AR1,P#1.0];
      L     6;	//Number of bytess to transfer
      T     LW [AR1,P#2.0];
      L     0;	//Type of data memory
      T     LW [AR1,P#4.0];
      L     DIW 0;
      SLD   3;
      L     P#I 0.0;
      +D;
      T     LD [AR1,P#6.0];
//Creation of a pointer to the target area
      LAR1  P##tempDST;	//Load initial address of destination pointer in AR1
      L     B#16#10;	//Load the ID for the ANY type
      T     LB [AR1,P#0.0];
      L     B#16#2;	//2=type of data is BYTE
      T     LB [AR1,P#1.0];
      L     6;	//Number of bytes to receive
      T     LW [AR1,P#2.0];
      L     0;	//Type of data memory
      T     LW [AR1,P#4.0];
      L     P##InputBuffer;
      T     LD [AR1,P#6.0];
//Trasfering data
      CALL  "BLKMOV" (
           SRCBLK                   := #tempSRC,
           RET_VAL                  := #tempINT,
           DSTBLK                   := #tempDST);
//Load saved registry value
      LAR1  #tempAR1;
      LAR2  #tempAR2;
NETWORK
TITLE = Mapping of the outputs
//Save registry value
      TAR1  #tempAR1;
      TAR2  #tempAR2;
//Creation of a pointer to the source area
      LAR1  P##tempSRC;	//Load initial address of source pointer in AR1
      L     B#16#10;	//Load the ID for the ANY type
      T     LB [AR1,P#0.0];
      L     B#16#2;	//2=type of data is BYTE
      T     LB [AR1,P#1.0];
      L     6;	//Number of bytess to transfer
      T     LW [AR1,P#2.0];
      L     0;	//Type of data memory
      T     LW [AR1,P#4.0];
      L     DIW 0;
      SLD   3;
      L     P#Q 0.0;
      +D;
      T     LD [AR1,P#6.0];
//Creation of a pointer to the target area
      LAR1  P##tempDST;	//Load initial address of destination pointer in AR1
      L     B#16#10;	//Load the ID for the ANY type
      T     LB [AR1,P#0.0];
      L     B#16#2;	//2=type of data is BYTE
      T     LB [AR1,P#1.0];
      L     6;	//Number of bytes to receive
      T     LW [AR1,P#2.0];
      L     0;	//Type of data memory
      T     LW [AR1,P#4.0];
      L     P##OutputBuffer;
      T     LD [AR1,P#6.0];
//Trasfering data
      CALL  "BLKMOV" (
           SRCBLK                   := #tempSRC,
           RET_VAL                  := #tempINT,
           DSTBLK                   := #tempDST);
//Load saved registry value
      LAR1  #tempAR1;
      LAR2  #tempAR2;
NETWORK
TITLE = Read job of header 1
      A     DIX 14.3;
      A     M 1.5;
      JCN   L006;
      L     DIB 18;
      L     1;
      +I;
      T     DIB 18;
L006: NOP   0;
//Select the header
      A     DIX 14.0;
      AN    DIX 15.0;
//UN    #Testa2.Lettura_Start
//UN    #Testa2.Scrittura_Start
      AN    DIX 14.3;
      S     DIX 14.3;
      R     DIX 8.4;
      JCN   L005;
      L     0;
      T     DIB 18;
L005: NOP   0;
//Check the header selected
      A     DIX 14.0;
      A     DIX 14.3;
      AN    DIX 2.4;
      AN    DIX 14.4;
      S     DIX 14.4;
//Start reading job
      A     DIX 14.0;
      A     DIX 14.4;
      A     DIX 2.7;
      A     DIX 2.0;
      AN    DIX 14.5;
      S     DIX 14.5;
      R     DIX 14.1;
      R     DIX 14.2;
      S     DIX 8.0;
      R     DIX 8.7;
      JC    L001;
      JU    L004;
L001: NOP   0;
      L     0;
      T     DIB 10;
      T     DIB 11;
      T     DIB 13;
      L     1;
      T     DIB 12;
      L     1;
      T     DIB 9;
L004: NOP   0;
//Read job ended with error
      A     DIX 14.0;
      A     DIX 14.5;
      A     DIX 2.1;
      A     DIX 2.3;
      O;
      A(;
      L     DIB 18;
      L     10;
      >=I;
      );
      R     DIX 14.3;
      R     DIX 14.4;
      R     DIX 14.5;
      R     DIX 8.0;
      R     DIX 14.0;
      S     DIX 14.2;
      JCN   L007;
      L     0;
      T     DIB 18;
L007: NOP   0;
//Read job ended without error
      A     DIX 14.0;
      A     DIX 14.5;
      A     DIX 2.1;
      A     DIX 2.2;
      R     DIX 14.3;
      R     DIX 14.4;
      R     DIX 14.5;
      R     DIX 8.0;
      R     DIX 14.0;
      S     DIX 14.1;
      JC    L002;
      JU    L003;
L002: L     DIB 3;
//T     #tempBYTE1
//L     #InputBuffer.Data1
//T     #tempBYTE2
//L     LW    36
      T     DIB 16;
L003: NOP   0;
NETWORK
TITLE = Write job of header 1
      A     DIX 15.3;
      A     M 1.5;
      JCN   L018;
      L     DIB 18;
      L     1;
      +I;
      T     DIB 18;
L018: NOP   0;
//Select the header
      A     DIX 15.0;
      AN    DIX 14.0;
//UN    #Testa2.Lettura_Start
//UN    #Testa2.Scrittura_Start
      AN    DIX 15.3;
      S     DIX 15.3;
      R     DIX 8.4;
      JCN   L015;
      L     0;
      T     DIB 18;
L015: NOP   0;
//Check the header selected
      A     DIX 15.0;
      A     DIX 15.3;
      AN    DIX 2.4;
      AN    DIX 15.4;
      S     DIX 15.4;
//Start writing job
      A     DIX 15.0;
      A     DIX 15.4;
      A     DIX 2.7;
      A     DIX 2.0;
      AN    DIX 15.5;
      S     DIX 15.5;
      R     DIX 15.1;
      R     DIX 15.2;
      S     DIX 8.0;
      R     DIX 8.7;
      JC    L011;
      JU    L012;
L011: NOP   0;
      L     0;
      T     DIB 10;
      T     DIB 11;
      T     DIB 13;
      L     1;
      T     DIB 12;
      L     2;
      T     DIB 9;
L012: NOP   0;
//Confirm write job in course
      A     DIX 15.0;
      A     DIX 15.5;
      A     DIX 2.1;
      A     DIX 2.5;
      AN    DIX 15.6;
      S     DIX 15.6;
      S     DIX 8.6;
      JC    L016;
      JU    L017;
L016: NOP   0;
      L     DIB 17;
//T     LW    36
//L     #tempBYTE1
      T     DIB 9;
//L     #tempBYTE2
//T     #OutputBuffer.StartAddress_L
L017: NOP   0;
//Write job ended with error
      A     DIX 15.0;
      A     DIX 15.6;
      A     DIX 2.1;
      A     DIX 2.3;
      O;
      A(;
      L     DIB 18;
      L     10;
      >=I;
      );
      R     DIX 15.3;
      R     DIX 15.4;
      R     DIX 15.5;
      R     DIX 15.6;
      R     DIX 8.0;
      R     DIX 8.6;
      R     DIX 15.0;
      S     DIX 15.2;
      JCN   L019;
      L     0;
      T     DIB 18;
L019: NOP   0;
//Write job ended without error
      A     DIX 15.0;
      A     DIX 15.6;
      A     DIX 2.1;
      A     DIX 2.2;
      R     DIX 15.3;
      R     DIX 15.4;
      R     DIX 15.5;
      R     DIX 15.6;
      R     DIX 8.0;
      R     DIX 8.6;
      R     DIX 15.0;
      S     DIX 15.1;
NETWORK
TITLE = Read job of header 2
      A     DIX 20.3;
      A     M 1.5;
      JCN   L026;
      L     DIB 24;
      L     1;
      +I;
      T     DIB 24;
L026: NOP   0;
//Select the header
      A     DIX 20.0;
      AN    DIX 21.0;
      AN    DIX 14.0;
      AN    DIX 15.0;
      AN    DIX 20.3;
      S     DIX 20.3;
      S     DIX 8.4;
      JCN   L025;
      L     0;
      T     DIB 24;
L025: NOP   0;
//Check the header selected
      A     DIX 20.0;
      A     DIX 20.3;
      A     DIX 2.4;
      AN    DIX 20.4;
      S     DIX 20.4;
//Start reading job
      A     DIX 20.0;
      A     DIX 20.4;
      A     DIX 2.7;
      A     DIX 2.0;
      AN    DIX 20.5;
      S     DIX 20.5;
      R     DIX 20.1;
      R     DIX 20.2;
      S     DIX 8.0;
      R     DIX 8.7;
      JC    L021;
      JU    L024;
L021: NOP   0;
      L     0;
      T     DIB 10;
      T     DIB 11;
      T     DIB 13;
      L     1;
      T     DIB 12;
      L     1;
      T     DIB 9;
L024: NOP   0;
//Read job ended with error
      A     DIX 20.0;
      A     DIX 20.5;
      A     DIX 2.1;
      A     DIX 2.3;
      O;
      A(;
      L     DIB 24;
      L     10;
      >=I;
      );
      R     DIX 20.3;
      R     DIX 20.4;
      R     DIX 20.5;
      R     DIX 8.0;
      R     DIX 20.0;
      S     DIX 20.2;
      JCN   L027;
      L     0;
      T     DIB 24;
L027: NOP   0;
//Read job ended without error
      A     DIX 20.0;
      A     DIX 20.5;
      A     DIX 2.1;
      A     DIX 2.2;
      R     DIX 20.3;
      R     DIX 20.4;
      R     DIX 20.5;
      R     DIX 8.0;
      R     DIX 20.0;
      S     DIX 20.1;
      JC    L022;
      JU    L023;
L022: L     DIB 3;
//T     #tempBYTE1
//L     #InputBuffer.Data1
//T     #tempBYTE2
//L     LW    36
      T     DIB 22;
L023: NOP   0;
NETWORK
TITLE = Write job of header 2
      A     DIX 21.3;
      A     M 1.5;
      JCN   L038;
      L     DIB 24;
      L     1;
      +I;
      T     DIB 24;
L038: NOP   0;
//Select the header
      A     DIX 21.0;
      AN    DIX 20.0;
      AN    DIX 14.0;
      AN    DIX 15.0;
      AN    DIX 21.3;
      S     DIX 21.3;
      S     DIX 8.4;
      JCN   L035;
      L     0;
      T     DIB 24;
L035: NOP   0;
//Check the header selected
      A     DIX 21.0;
      A     DIX 21.3;
      A     DIX 2.4;
      AN    DIX 21.4;
      S     DIX 21.4;
//Start writing job
      A     DIX 21.0;
      A     DIX 21.4;
      A     DIX 2.7;
      A     DIX 2.0;
      AN    DIX 21.5;
      S     DIX 21.5;
      R     DIX 21.1;
      R     DIX 21.2;
      S     DIX 8.0;
      R     DIX 8.7;
      JC    L031;
      JU    L032;
L031: NOP   0;
      L     0;
      T     DIB 10;
      T     DIB 11;
      T     DIB 13;
      L     1;
      T     DIB 12;
      L     2;
      T     DIB 9;
L032: NOP   0;
//Confirm write job in course
      A     DIX 21.0;
      A     DIX 21.5;
      A     DIX 2.1;
      A     DIX 2.5;
      AN    DIX 21.6;
      S     DIX 21.6;
      S     DIX 8.6;
      JC    L036;
      JU    L037;
L036: NOP   0;
      L     DIB 23;
//T     LW    36
//L     #tempBYTE1
      T     DIB 9;
//L     #tempBYTE2
//T     #OutputBuffer.StartAddress_L
L037: NOP   0;
//Write job ended with error
      A     DIX 21.0;
      A     DIX 21.6;
      A     DIX 2.1;
      A     DIX 2.3;
      O;
      A(;
      L     DIB 24;
      L     10;
      >=I;
      );
      R     DIX 21.3;
      R     DIX 21.4;
      R     DIX 21.5;
      R     DIX 21.6;
      R     DIX 8.0;
      R     DIX 8.6;
      R     DIX 21.0;
      S     DIX 21.2;
      JCN   L039;
      L     0;
      T     DIB 24;
L039: NOP   0;
//Write job ended without error
      A     DIX 21.0;
      A     DIX 21.6;
      A     DIX 2.1;
      A     DIX 2.2;
      R     DIX 21.3;
      R     DIX 21.4;
      R     DIX 21.5;
      R     DIX 21.6;
      R     DIX 8.0;
      R     DIX 8.6;
      R     DIX 21.0;
      S     DIX 21.1;
NETWORK
TITLE = Mapping of the outputs
//Save registry value
      TAR1  #tempAR1;
      TAR2  #tempAR2;
//Creation of a pointer to the source area
      LAR1  P##tempSRC;	//Load initial address of source pointer in AR1
      L     B#16#10;	//Load the ID for the ANY type
      T     LB [AR1,P#0.0];
      L     B#16#2;	//2=type of data is BYTE
      T     LB [AR1,P#1.0];
      L     6;	//Number of bytess to transfer
      T     LW [AR1,P#2.0];
      L     0;	//Type of data memory
      T     LW [AR1,P#4.0];
      L     P##OutputBuffer;
      T     LD [AR1,P#6.0];
//Creation of a pointer to the target area
      LAR1  P##tempDST;	//Load initial address of destination pointer in AR1
      L     B#16#10;	//Load the ID for the ANY type
      T     LB [AR1,P#0.0];
      L     B#16#2;	//2=type of data is BYTE
      T     LB [AR1,P#1.0];
      L     6;	//Number of bytes to receive
      T     LW [AR1,P#2.0];
      L     0;	//Type of data memory
      T     LW [AR1,P#4.0];
      L     DIW 0;
      SLD   3;
      L     P#Q 0.0;
      +D;
      T     LD [AR1,P#6.0];
//Trasfering data
      CALL  "BLKMOV" (
           SRCBLK                   := #tempSRC,
           RET_VAL                  := #tempINT,
           DSTBLK                   := #tempDST);
//Load saved registry value
      LAR1  #tempAR1;
      LAR2  #tempAR2;
END_FUNCTION_BLOCK

